FUNCTION "ASW_MAL1S032Ctrl" : VOID
TITLE =MAL1S032 Section control: LINE 1 SEC 32 KILN 1
//COPYRIGHT:    (C) 2009 BY  BUHLER AG
//                           CH-9240 UZWIL  SWITZERLAND
//
//PRODUCT:      WinCoS_BIW01_09
//
//TITLE:        LINE 1 SEC 32 KILN 1
//                 Section control
//
//--------------------------------------------------------------------------------
//
//IDENT:        AUTHOR:             DEPT:                              DATE:
//
//P01_FC832.1.0 K.Renz              CSB41                              09.Okt.2009
//              1st Release
//
//--------------------------------------------------------------------------------
//
//PURPOSE:
//
//REFERENCES : GCSOSMAN
//
//--------------------------------------------------------------------------------
//
//
//0000 to 0999: Main Functions
//              0 =Main Function Cylic
//              1 =Main Function Coldstart/Newstart
//              2 =Main Function Warm Start
AUTHOR : KR
FAMILY : USW
VERSION : 9.9


VAR_INPUT
  InCode : INT ;
END_VAR
VAR_TEMP
  tmpStartNext : BOOL ;	//Condition to Start next element
  tmpFlagFault : BOOL ;	//Flag mechanical fault
  tmpEnableFeed : BOOL ;
  tmpStartScale : BOOL ;
  tmpStartLiqScale : BOOL ;	//Enable to Start Lipquid Scale
  tmpSndBin : INT ;
  tmpRcvBin : INT ;
  tmpBool : BOOL ;
  tmpByte : BYTE ;
  tmpWord : WORD ;
  tmpDWord : DWORD ;
  tmpInt : INT ;
  tmpRET : INT ;
  tmpDInt : DINT ;
  tmpCyclusTime : DINT ;
  tmpWetSteep : BOOL ;
END_VAR
BEGIN
NETWORK
TITLE =
//=================================================
//=================================================
//S T A R T   M A I N   F U N C T I O N
//=================================================
//=================================================
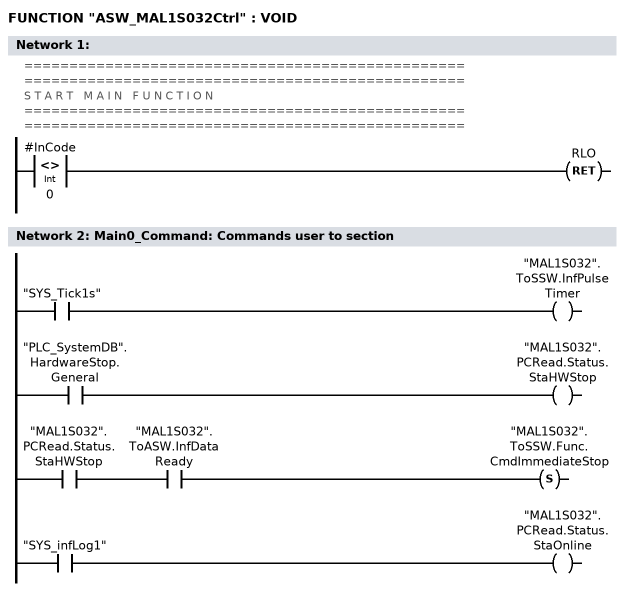
      L     #InCode;
      L     0;
      <>I   ;
      BEB   ;

NETWORK
TITLE =Main0_Command: Commands user to section

      NOP   0;
//-Tick 1 second---
      U     "SYS_Tick1s";
      =     "MAL1S032".ToSSW.InfPulseTimer;
//-Hardware stop---
      U     "PLC_SystemDB".HardwareStop.General;
      =     "MAL1S032".PCRead.Status.StaHWStop;
      U     "MAL1S032".PCRead.Status.StaHWStop;
      U     "MAL1S032".ToASW.InfDataReady;
      S     "MAL1S032".ToSSW.Func.CmdImmediateStop;
//-Online---
      U     "SYS_infLog1";
      =     "MAL1S032".PCRead.Status.StaOnline;
NETWORK
TITLE =ASW_UC: User commands to section

      NOP   0;
//-Additional user commands---
//-GP standard commands---
      AUF   "MAL1S032";
      L     L#0; // Enter the differenz of the target weight and prestop weight
      T     "MAL1S032".VarTemp.InOutValue3; // Prestop weight
      CALL "STD_LineSecStdSub" (
           InCode                   := 2001);// Section function: Standard section commands

//-Condition CmdSequenzStop---
      U     "MAL1S032".ToSSW.Func.CmdSequenzStop;
//      S     "MAL1S032".ToSSW.Func.CmdSequenzStop
      R     "MAL1S032".ToSSW.Func.CmdSequenzStop;
//-Extended section commands---
//      AUF   "MAL1S032"
//      CALL  "STD_LineSecStdSub"
//       InCode:=2002                     // Section function: Extended section commands
//-Status from pulse commands---
      CLR   ;
      =     "MAL1S032".PCRead.ExtFuncOn.Pulse00OverrideLL;
      =     "MAL1S032".PCRead.ExtFuncOn.Pulse01;
      =     "MAL1S032".PCRead.ExtFuncOn.Pulse02;
      =     "MAL1S032".PCRead.ExtFuncOn.Pulse03;
      =     "MAL1S032".PCRead.ExtFuncOn.Pulse04;
      =     "MAL1S032".PCRead.ExtFuncOn.Pulse05;
      =     "MAL1S032".PCRead.ExtFuncOn.Pulse06;
      =     "MAL1S032".PCRead.ExtFuncOn.Pulse07;
//
NETWORK
TITLE =Main0_Dest: Destination
//99 = Undefined Condition
// 0 = Wait to Loading
// 1 = Loading
// 2 = Process Aktive
// 3 = Unloading
// 4 = Cleaning
// 5 = Finish Unloading
// 6 = Process End
// 7 = Cooling Active
// 8 = Wait to Unloading
// 9 =
//10 = Wait for Start Loading
//11 = Start process is not possible! First loading round is not closed!
//12 = Wait for Start Process
//13 = Can not be unloaded! Same batch in previous section!
//14 = Turning is not possible! Srew is not in position!
//15 = Cleaning not finished!
//16 = Process aktive and wait for water! Water not filled!
//17 = Spraying is not possible! Wait for water!
//18 = Cleaning is not possible! Wait for water!
//19 = Automatic function obstructs by active ILO-Mode!
//20 = Automatic startup is breacked! Wait for continue!
//21 = Wait for release unloading!
//22 = Brennerluft zu kalt!   // NEU
      L     99; // Undefined condition

      U     "MAL1S032".PCRead.Step.StPassive;
      UN    "MAL1S032".ToASW.InfDataReady;
      O     ;
      U     "MAL1S032".PCRead.Step.StIdling;
      UN    "MAL1S032".ToASW.InfDataReady;
      SPBN  M300;
      L     0; // Wait for loading
      SPA   M030;
M300: NOP   0;

      U     "MAL1S032".PCRead.Step.StWait;
      U     "MAL1S032".ToASW.InfDataReady;
      SPBN  M310;
      L     10; // Wait for start loading
      SPA   M030;
M310: NOP   0;

      U     "MAL1S032".ToASW.InfDataReady;
      UN    "MAL1S032".PCRead.Step.StWait;
      UN    "MAL1S032".PCRead.Fault.EsMech;
//    UN    "MAL1S006".PCRead.Status.StaAutostart
      U     DB832.DBX  123.0;
      U     DB832.DBX  123.1;
      SPBN  M320;
      L     20; // Automatic startup is breacked! Wait for continue!
      SPA   M030;
M320: NOP   0;

      U     "MAL1S032".PCWrite.ExtFuncOn.StartProcess;
      L     S5T#30S;
      SA    T     86;
      U     T     86;

      U     "MAL1S032".PCRead.Step.StActive;
      U     "MAL1S032Par".Par.FlagFunction_1.StepLoading;
      UN    "MAL1S032Par".Par.FlagProcess.ProcessActive;
      U     "MAL1S032Par".Par.FlagFunction_1.LoadEnd;
      UN    "MAL1S032Par".Par.FlagFunction_1.LoadFirstPartEnd;
// Prozess-Start erst moeglich wenn Darre 2 Schritt 3 beendet hat oder nicht aktiv ist!!
      U(    ;
      U(    ;
      L     "MAL1S033Par".Par.ParIntMachine.ActualStep;
      L     4;
      >=I   ;
      )     ;
      ON    "MAL1S033Par".Par.FlagProcess.ProcessActive;
      )     ;

      SPBN  M311;
      L     11; // Start process is not possible! First loading round is not closed!
      SPA   M030;
M311: NOP   0;

      U     "MAL1S032".ToASW.InfDataReady;
      U(    ;
      O     "MAL1S032".PCRead.Step.StActive;
      O     "MAL1S032".PCRead.Step.StReady;
      )     ;
      U     "MAL1S032Par".Par.FlagFunction_1.FinishLoading;
      U     "G266M".A_3111_MXZ41MA.A_3111_BZS43.StTrue; // sensor zero point
      UN    "MAL1S032Par".Par.FlagProcess.ProcessActive; // Process active
      SPBN  M312;
      L     12; // Wait for start process
      SPA   M030;
M312: NOP   0;

      U     "MAL1S032".ToASW.InfDataReady;
      U     "MAL1S032Par".Par.FlagFunction_1.StepLoading;
      UN    "MAL1S032Par".Par.FlagFunction_1.FinishLoading;
      UN    "MAL1S032Par".Par.FlagProcess.ProcessActive;
      SPBN  M301;
      L     1; // Loading
      SPA   M030;
M301: NOP   0;

      U     "MAL1S032Par".Par.FlagProcess.TurningFloor;
      UN(   ;
      U     "G265M".A_3111_MXZ21_31MA.A_3111_BZS33.InpTrue;
      U     "G265M".A_3111_MXZ21_31MA.A_3111_BZS23.InpTrue;
      )     ;
      SPBN  M314;
      L     14; // Turning is not possible! Srew is not in position!
      SPA   M030;
M314: NOP   0;

      U     "SYS_infLog0";
      SPBN  M317;
      L     17; // Spraying is not possible! Wait for water!
      SPA   M030;
M317: NOP   0;

      U     "G266M".Gr.InManual; // FLOOR DRIVES KILNINGBOX 1
      UN    "G266M".Gr.VarFault; // FLOOR DRIVES KILNINGBOX 1
      U     "G266M".A_3111_MXZ41MA.Ma.StStopped; // FLOOR DRIVES KILNINGBOX 1
      U     "MAL1S032Par".Par.FlagFunction_1.TurningStart;
      U     "MAL1S032Par".Par.FlagProcess.TurningFloor;
      U     "MAL1S032".ToASW.InfDataReady;
      SPBN  M319;
      L     19; // Automatic function obstructs by active ILO-Mode!
      SPA   M030;
M319: NOP   0;

      U     "MAL1S032".Gr.OutSelected[303]; //-->G303M Defroster Flaps Kilningbox
      UN    "MAL1S032Par".Par.FlagProcess2.Schaltp_5;
      U     "MAL1S032Par".Par.FlagProcess.ProcessActive;
      UN    "MAL1S032Par".Par.FlagProcess.Cooling_Activ;
      SPBN  M322;
      L     22; // Brennerluft zu kalt!
      SPA   M030;
M322: NOP   0;

      U     "MAL1S032Par".Par.FlagProcess.ProcessActive;
      UN    "MAL1S032Par".Par.FlagProcess.Cooling_Activ;
      SPBN  M302;
      L     2; // Process aktive
      SPA   M030;
M302: NOP   0;

      U     "MAL1S032".ToASW.InfDataReady;
      UN    "MAL1S034".PCRead.State.StFeeding;
      U     "MAL1S032Par".Par.FlagFunction_1.StepUnloading;
      UN    "MAL1S032Par".Par.FlagFunction_1.FinishUnloading;
      SPBN  M321;
      L     21; // Wait for release unloading!
      SPA   M030;
M321: NOP   0;

      U     "MAL1S032".ToASW.InfDataReady;
      U     "MAL1S032Par".Par.FlagFunction_1.StepUnloading;
      SPBN  M303;
      L     3; // Unloading
      SPA   M030;
M303: NOP   0;

      U     "SYS_infLog0";
      SPBN  M315;
      L     15; // Cleaning not finished!
      SPA   M030;
M315: NOP   0;

      U     "SYS_infLog0";
      SPBN  M318;
      L     18; // Cleaning is not possible! Wait for water!
      SPA   M030;
M318: NOP   0;

      U     "MAL1S032".ToASW.InfDataReady;
      U     "MAL1S032Par".Par.FlagFunction_1.StepCleaning;
      UN    "MAL1S032Par".Par.FlagFunction_1.FinishCleaning;
      SPBN  M304;
      L     4; // Cleaning
      SPA   M030;
M304: NOP   0;

      U     "MAL1S032".ToASW.InfDataReady;
      U     "MAL1S032Par".Par.FlagFunction_1.FinishUnloading;
      UN    "MAL1S032Par".Par.FlagFunction_1.StepCleaning;
      UN    "MAL1S032Par".Par.FlagFunction_1.FinishCleaning;
      SPBN  M305;
      L     5; // Finish unloading
      SPA   M030;
M305: NOP   0;

      U     "SYS_infLog0";
      SPBN  M306;
      L     6; // Process End
      SPA   M030;
M306: NOP   0;

      U     "MAL1S032Par".Par.FlagProcess.ProcessActive; // Process active
      U     "MAL1S032Par".Par.FlagProcess.Cooling_Activ; // Cooling
      SPBN  M307;
      L     7; // Cooling Active
      SPA   M030;
M307: NOP   0;

      U     "MAL1S032".ToASW.InfSameBatchPrevSec;
      U     "MAL1S032".ToASW.InfDataReady;
      U     "MAL1S032Par".Par.FlagProcess.ProcessEnd;
      UN    "MAL1S032Par".Par.FlagProcess.ProcessActive;
      UN    "MAL1S032Par".Par.FlagFunction_1.StepLoading;
      UN    "MAL1S032Par".Par.FlagFunction_1.StepUnloading;
      SPBN  M313;
      L     13; // Can not be unloaded! Same batch in previous section!
      SPA   M030;
M313: NOP   0;

      U     "MAL1S032".ToASW.InfDataReady;
      UN    "MAL1S032".ToASW.InfSameBatchPrevSec;
      U     "MAL1S032Par".Par.FlagProcess.ProcessEnd;
      UN    "MAL1S032Par".Par.FlagProcess.ProcessActive;
      UN    "MAL1S032Par".Par.FlagFunction_1.StepUnloading;
      UN    "MAL1S032Par".Par.FlagFunction_1.FinishUnloading;
      UN    "MAL1S032Par".Par.FlagFunction_1.StepCleaning;
      UN    "MAL1S032Par".Par.FlagFunction_1.FinishCleaning;
      SPBN  M308;
      L     8; // Wait for Unloading
      SPA   M030;
M308: NOP   0;

      U     "SYS_infLog0";
      SPBN  M316;
      L     16; // Process aktive and wait for water! Water not filled!
      SPA   M030;
M316: NOP   0;

M030: T     "MAL1S032Par".SectionStatus;


NETWORK
TITLE =Main0_Next: Ready for next batch

      ON    "MAL1S032".ToASW.InfDataReady;
      =     "MAL1S032".ToSSW.InfReadyForNewBatch;
NETWORK
TITLE =Main0_Control: Control section

      NOP   0;
//-Process commands from PCS---
      AUF   "MAL1S032";
      CALL "GCS7_SecCtrlMain" (// Methode O_Section
           CODE                     := 7);
//-Process commands from user---
      AUF   "MAL1S032";
      CALL "GCS7_SecCtrlMain" (// Methode Control
           CODE                     := 0);
//-Process section step---
      AUF   "MAL1S032";
      CALL "GCS7_SecCtrlMain" (// Methode Step_execute
           CODE                     := 2);
      AUF   "MAL1S032";
      CALL "GCS7_SecCtrlMain" (// Methode Step_transition
           CODE                     := 3);
//-Process section state---
      AUF   "MAL1S032";
      CALL "GCS7_SecCtrlMain" (// Methode State
           CODE                     := 4);

NETWORK
TITLE =Main0_Init: Init

      UN    "MAL1S032".ToASW.Transition.ToWait;
      UN    "MAL1S032".ToASW.CmdNewBatch;
      SPB   in00;
//-User initialization---
      AUF   "MAL1S032";
//
//-Section function: Init ---
      AUF   "MAL1S032";
      CALL "STD_LineSecStdSub" (
           InCode                   := 2003);// Section function: Init
//
//-Group interface---
//
//-Initialise bin objects---
//
//-Emptying job---
      U     "MAL1S032".JobAc.StaBatch.StaEmptyingBatch;
      S     "MAL1S032".PCRead.Status.StaLoaded;
//
//-Error Batch---
//
in00: NOP   0;

NETWORK
TITLE =ASW_VB: Various functions before bin control

      NOP   0;
//
//-Update staSameSndRcv in sender binlist---
NETWORK
TITLE =Main0_GrEMM: Enable manual mode
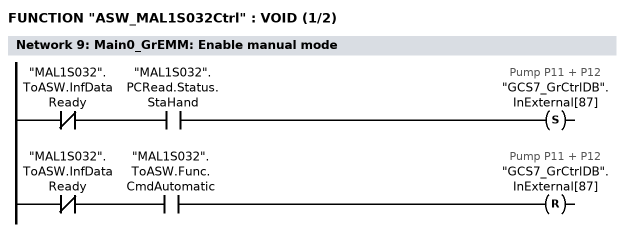

      UN    "MAL1S032".ToASW.InfDataReady;
      U     "MAL1S032".PCRead.Status.StaHand;
      S     "GCS7_GrCtrlDB".InExternal[87]; // Pump P11 + P12

      UN    "MAL1S032".ToASW.InfDataReady;
      U     "MAL1S032".ToASW.Func.CmdAutomatic;
      R     "GCS7_GrCtrlDB".InExternal[87]; // Pump P11 + P12

NETWORK
TITLE =Main0_GrNRS: Not Relevant for started / Fault
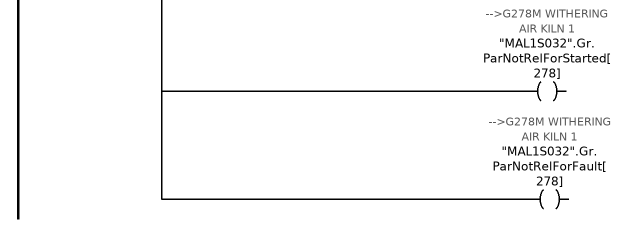

      NOP   0;
      SET   ;
      =     "MAL1S032".Gr.ParNotRelForStarted[1]; //-->G001G Power supply circuit +C11
      =     "MAL1S032".Gr.ParNotRelForFault[1]; //-->G001G Power supply circuit +C11
      =     "MAL1S032".Gr.ParNotRelForStarted[2]; //-->G002G Contactor panel power supply 1
      =     "MAL1S032".Gr.ParNotRelForFault[2]; //-->G002G Contactor panel power supply 1
      =     "MAL1S032".Gr.ParNotRelForStarted[3]; //-->G003G PLC monitoring
      =     "MAL1S032".Gr.ParNotRelForFault[3]; //-->G003G PLC monitoring
      =     "MAL1S032".Gr.ParNotRelForStarted[26]; // -->G026G Alarm horns
      =     "MAL1S032".Gr.ParNotRelForFault[26]; // -->G026G Alarm horns
      =     "MAL1S032".Gr.ParNotRelForStarted[269]; //-->G269M Temperature Mes.  Kilningbox 1
      =     "MAL1S032".Gr.ParNotRelForFault[269]; //-->G269M Temperature Mes.  Kilningbox 1

      U     "MAL1S032Par".Par.FlagFunction_1.StepLoading;
      =     "MAL1S032".Gr.ParNotRelForStarted[271]; //-->G271M FAN KILN 1
      =     "MAL1S032".Gr.ParNotRelForFault[271]; //-->G271M FAN KILN 1
      =     "MAL1S032".Gr.ParNotRelForStarted[272]; //-->G272M FRESH AIR LOUVER KILN 1
      =     "MAL1S032".Gr.ParNotRelForFault[272]; //-->G272M FRESH AIR LOUVER KILN 1
      =     "MAL1S032".Gr.ParNotRelForStarted[273]; //-->G273M RECYCLING AIR LOUVER KILN 1
      =     "MAL1S032".Gr.ParNotRelForFault[273]; //-->G273M RECYCLING AIR LOUVER KILN 1
      =     "MAL1S032".Gr.ParNotRelForStarted[274]; //-->G274M EXHAUST AIR LOUVER KILN 1
      =     "MAL1S032".Gr.ParNotRelForFault[274]; //-->G274M EXHAUST AIR LOUVER KILN 1
      =     "MAL1S032".Gr.ParNotRelForStarted[275]; //-->G275M LOUVER HEATING GLASS TUBE HEAT EXCHANGER
      =     "MAL1S032".Gr.ParNotRelForFault[275]; //-->G275M LOUVER HEATING GLASS TUBE HEAT EXCHANGER
      =     "MAL1S032".Gr.ParNotRelForStarted[276]; //-->G276 MHEATING KILN 1
      =     "MAL1S032".Gr.ParNotRelForFault[276]; //-->G276M HEATING KILN 1
      =     "MAL1S032".Gr.ParNotRelForStarted[277]; //-->G277M LOUVER AIR HEATER 1 FOR KILN 1
      =     "MAL1S032".Gr.ParNotRelForFault[277]; //-->G277M LOUVER AIR HEATER 1 FOR KILN 1
      =     "MAL1S032".Gr.ParNotRelForStarted[278]; //-->G278M WITHERING AIR KILN 1
      =     "MAL1S032".Gr.ParNotRelForFault[278]; //-->G278M WITHERING AIR KILN 1

      NOP   0;

NETWORK
TITLE =Main0_GrSelection: Group selection
// List of the used objects in the section
// ==========================
// G021G       GENERAL ELEMENTS KILN 1
// G284M       BELT CONVEYOR 7100 KILN
// G261M       BELT CONVEYOR 7200 KILN
// G262M       BELT CONVEYOR 7300 KILN
// G263M       BELT CONVEYOR 7301 KILN
// G264M       BELT CONVEYOR 7400 KILN
// G265M       LIFTING DEVICE KILN 1
// G266M       TRAVELLING DRIVE KILN 1
// G267M       UNLOADING / LOADING SCREW KILN 1
// G268M       DISCHARGE DOOR KILN 1
// G269M       TEMPERATURE MES. KILN 1
// G270M       AIR SHUT SLIDE KILN 1
// G271M       FAN KILN 1
// G272M       FRESH AIR LOUVER KILN 1
// G273M       RECYCLING AIR LOUVER KILN 1
// G274M       EXHAUST AIR LOUVER KILN 1
// G275M       LOUVER HEATING GLASS TUBE HEAT EXCHANGER
// G276M       HEATING KILN 1
// G277M       LOUVER AIR HEATER 1 FOR KILN 1
// G278M       WITHERING AIR KILN 1
// G279M       HEATING KILN 1 + 2
// G280M       CHAIN CONVEYOR 9001 KILN 1
// G281M       ELEVATOR 9002 AFTER KILN
// G282M       FLAP BOX 9008
// G283M       CULM BATCH BIN 9005
//
      NOP   0;
//-Condition for preselection---
      U     "MAL1S032".ToASW.InfDataReady;
      SPB   GS01;
//-Deselect groups ---
      CALL "GCS7_GrpCtrlMain" , "GCS7_GrCtrlDBTmp" (// GrCtr.Methode Deselect
           Code                     := 3,
           Sec                      := "MAL1S032".Gr);
      SPA   GS02;
//-Select groups ---
GS01: NOP   0;
//-Prepare for preselection ---
      CALL "GCS7_GrpCtrlMain" , "GCS7_GrCtrlDBTmp" (// GrCtr.Methode Init Preselection
           Code                     := 1,
           Sec                      := "MAL1S032".Gr);
//
//
//-Preselect used groups --
      SET   ;
      S     "MAL1S032".Gr.InPreselect[21]; //-->G021G GENERAL ELEMENTS KILN 1
      S     "MAL1S032".Gr.InPreselect[269]; //-->G269M TEMPERATURE MES. KILN 1

//--- Option
      U     "MAL1S032".PCRead.Step.StActive; // Loading
      O     "MAL1S032".PCRead.Step.StReady; // Process active
      U(    ;
      L     "G269M".A_3191_BTE11.OutValuePc; // AIR TEMPERATURE OUTSIDE
      L     1500; // 15.00°C
      <=I   ;
      )     ;
      UN(   ;
      U     "MAL1S032Par".Par.FlagProcess2.Schaltp_15;
      U     "MAL1S032Par".Par.FlagProcess2.Schaltp_70;
      )     ;
      U     "SYS_infLog0"; // Keine Freigabe!!
      S     "MAL1S032".Gr.InPreselect[276]; //-->G276M HEATING KILN 1
      S     "MAL1S032".Gr.InPreselect[277]; //-->G277M LOUVER AIR HEATER 1 FOR KILN 1
      S     "MAL1S032".Gr.InPreselect[275]; //-->G275M LOUVER HEATING GLASS TUBE HEAT EXCHANGER

// Oeffnen und Schliessen der Defroster-Klappe
      U     "G275M".USW8; // Defrosterklappe AUF
      S     "MAL1S032".Gr.InPreselect[275]; //-->G275M LOUVER HEATING GLASS TUBE HEAT EXCHANGER

//------------------------------Loading kilningbox-----------------------------------
      U     "MAL1S032".PCRead.Step.StActive;
      U     "MAL1S032Par".Par.FlagFunction_1.StepLoading; // Step loading
      S     "MAL1S032".Gr.InPreselect[265]; //-->G265M LIFTING DEVICE KILN 1

      U     "MAL1S032".PCRead.Step.StActive;
      U     "MAL1S032Par".Par.FlagFunction_1.StepLoading; // Step loading
      UN    "MAL1S032Par".Par.FlagFunction_1.FinishLoading; // start process kilning
      S     "MAL1S032".Gr.InPreselect[266]; //-->G266M TRAVELLING DRIVE KILN 1
      S     "MAL1S032".Gr.InPreselect[267]; //-->G267M UNLOADING / LOADING SCREW KILN 1
      S     "MAL1S032".Gr.InPreselect[268]; //-->G268M DISCHARGE DOOR KILN 1
      S     "MAL1S032".Gr.InPreselect[270]; //-->G270M AIR SHUT SLIDE KILN 1
      S     "MAL1S032".Gr.InPreselect[284]; //-->G284M BELT CONVEYOR 7100 KILN
      S     "MAL1S032".Gr.InPreselect[261]; //-->G261M BELT CONVEYOR 7200 KILN
      S     "MAL1S032".Gr.InPreselect[262]; //-->G262M BELT CONVEYOR 7300 KILN
      S     "MAL1S032".Gr.InPreselect[263]; //-->G263M BELT CONVEYOR 7301 KILN
      S     "MAL1S032".Gr.InPreselect[264]; //-->G264M BELT CONVEYOR 7400 KILN

//----------------------------Loading kilningbox finish------------------------------
      U     "MAL1S032".PCRead.Step.StActive;
      O     "MAL1S032".PCRead.Step.StReady;
      U     "MAL1S032Par".Par.FlagProcess.ProcessActive;
      U(    ;
      UN    "G265M".A_3111_MXZ21_31MA.Ma.OutAdjustedLeft;
      ON    "G265M".A_3111_MXZ21_31MA.Ma.OutAdjustedRight;
      )     ;
      S     "MAL1S032".Gr.InPreselect[265]; //-->G265M LIFTING DEVICE KILN 1
//
      U(    ;
      U     "MAL1S032Par".Par.FlagProcess.ProcessActive;
      UN    "MAL1S032Par".Par.FlagFunction_1.StepLoading;
      O     "MAL1S032".PCRead.Step.StReady;
      )     ;
      U     "MAL1S032Par".Par.FlagProcess.ProcessActive;
      U     "MAL1S032Par".Par.FlagProcess.TurningFloor;
      U     "MAL1S032Par".Par.FlagFunction_1.TurningStart;
      S     "MAL1S032".Gr.InPreselect[266]; //-->G266M TRAVELLING DRIVE KILN 1

// Glaettungfahrt zur Parkposition bei Beladen Ende
      U     "MAL1S032Par".Par.FlagProcess.ProcessActive;
      U     "MAL1S032Par".Par.FlagMachine.ImpulsNullstellung;
      S     "MAL1S032".Gr.InPreselect[265]; //-->G265M LIFTING DEVICE KILN 1
      S     "MAL1S032".Gr.InPreselect[266]; //-->G266M TRAVELLING DRIVE KILN 1
      S     "MAL1S032".Gr.InPreselect[267]; //-->G267M UNLOADING / LOADING SCREW KILN 1

//-Cleaning conveyance after loading---
      UN    "MAL1S032Par".Par.FlagFunction_1.StepLoading;
      U     "MAL1S032".PCRead.Step.StReady;
      U     "MAL1S032Par".Par.FlagFunction_0.TimeCleanConvRun;
      S     "MAL1S032".Gr.InPreselect[284]; //-->G284M BELT CONVEYOR 7100 KILN
      S     "MAL1S032".Gr.InPreselect[261]; //-->G261M BELT CONVEYOR 7200 KILN
      S     "MAL1S032".Gr.InPreselect[262]; //-->G262M BELT CONVEYOR 7300 KILN
      S     "MAL1S032".Gr.InPreselect[263]; //-->G263M BELT CONVEYOR 7301 KILN
      S     "MAL1S032".Gr.InPreselect[264]; //-->G264M BELT CONVEYOR 7400 KILN


//-------------------------------Process kilning-------------------------------------
      U     "MAL1S032".PCRead.Step.StActive;
      O     "MAL1S032".PCRead.Step.StReady;
      U     "MAL1S032Par".Par.FlagProcess.ProcessActive; // Process active
      S     "MAL1S032".Gr.InPreselect[268]; //-->G268M DISCHARGE DOOR KILN 1
      S     "MAL1S032".Gr.InPreselect[270]; //-->G270M AIR SHUT SLIDE KILN 1
      S     "MAL1S032".Gr.InPreselect[271]; //-->G271M FAN KILN 1

      U     "MAL1S032".PCRead.Step.StActive;
      O     "MAL1S032".PCRead.Step.StReady;
      U     "MAL1S032Par".Par.FlagProcess.ProcessActive; // Process active
      O     ;
      U     "MAL1S032Par".Par.FlagProcess.ProcessEnd;
      UN    "MAL1S032Par".Par.FlagProcess.ProcessActive;
      UN    "GCS7_GrCtrlDB".InStopped[271]; //-->G271M FAN KILN 1
      S     "MAL1S032".Gr.InPreselect[273]; //-->G273M RECYCLING AIR LOUVER KILN 1
      S     "MAL1S032".Gr.InPreselect[278]; //-->G278M WITHERING AIR KILN 1

      U     "MAL1S032".PCRead.Step.StActive;
      O     "MAL1S032".PCRead.Step.StReady;
      U     "MAL1S032Par".Par.FlagProcess.ProcessActive;
      UN    "MAL1S032Par".Par.FlagProcess.Cooling_Activ;
      S     "MAL1S032".Gr.InPreselect[276]; //-->G276M HEATING KILN 1
      S     "MAL1S032".Gr.InPreselect[277]; //-->G277M LOUVER AIR HEATER 1 FOR KILN 1
      S     "MAL1S032".Gr.InPreselect[279]; //-->G279M HEATING KILN 1 + 2

//--------------------------Kuehlluft-Klappenregelung EIN----------------------------
      U     "MAL1S032".PCRead.Step.StActive;
      O     "MAL1S032".PCRead.Step.StReady;
      U     "MAL1S032Par".Par.FlagProcess.ProcessActive;
      UN    "MAL1S032Par".Par.FlagProcess.Cooling_Activ;
      U     "G272M".USW8; // Klappenregelung Ein
      S     "MAL1S032".Gr.InPreselect[272]; //-->G272M FRESH AIR LOUVER KILN 1

//-------------------------------Process Cooling--------------------------------------
      U     "MAL1S032".PCRead.Step.StActive;
      O     "MAL1S032".PCRead.Step.StReady;
      U     "MAL1S032Par".Par.FlagProcess.ProcessActive;
      U     "MAL1S032Par".Par.FlagProcess.Cooling_Activ;
      O     ;
      U     "MAL1S032Par".Par.FlagProcess.ProcessEnd;
      UN    "MAL1S032Par".Par.FlagProcess.ProcessActive;
      UN    "GCS7_GrCtrlDB".InStopped[271]; //-->G271M FAN KILN 1
      S     "MAL1S032".Gr.InPreselect[272]; //-->G272M FRESH AIR LOUVER KILN 1
      S     "MAL1S032".Gr.InPreselect[277]; //-->G277M LOUVER AIR HEATER 1 FOR KILN 1

//---------------------------Unloading kilning box------------------------------------
      U     "MAL1S032".PCRead.Step.StEmptying;
      U     "MAL1S032Par".Par.FlagFunction_1.StepUnloading; // Step unloading
      U     "MAL1S034".PCRead.State.StFeeding;
      S     "MAL1S032".Gr.InPreselect[268]; //-->G268M DISCHARGE DOOR KILN 1
//
      U     "MAL1S032".PCRead.Step.StEmptying;
      U     "MAL1S032Par".Par.FlagFunction_1.StepUnloading; // Step unloading
      U     "MAL1S034".PCRead.State.StFeeding;
      U     "G268M".Gr.OutEnablePrevGr; //-->G268M DISCHARGE DOOR KILN 1
      S     "MAL1S032".Gr.InPreselect[265]; //-->G265M LIFTING DEVICE KILN 1
//
      U     "MAL1S032".PCRead.Step.StEmptying;
      U     "MAL1S032Par".Par.FlagFunction_1.StepUnloading; // Step unloading
//      UN    "MAL1S032".PCRead.Status.StaTransferOffASW
      U     "G268M".Gr.OutEnablePrevGr; //-->G268M DISCHARGE DOOR KILN 1
      UN    "MAL1S032Par".Par.FlagFunction_1.FinishUnloading;
      U     "MAL1S034".PCRead.State.StFeeding;
      S     "MAL1S032".Gr.InPreselect[267]; //-->G267M UNLOADING / LOADING SCREW KILN 1
//
      U     "MAL1S032".PCRead.Step.StEmptying;
      U     "MAL1S032Par".Par.FlagFunction_1.StepUnloading; // Step unloading
      U     "MAL1S034".PCRead.State.StFeeding;
      UN    "MAL1S032".PCRead.Status.StaTransferOffASW;
      U     "G268M".Gr.OutEnablePrevGr; //-->G268M DISCHARGE DOOR KILN 1
      U     "G267M".Gr.OutEnablePrevGr; //-->G267M UNLOADING / LOADING SCREW KILN 1
      UN    "MAL1S032Par".Par.FlagFunction_0.ScrewAboveProductLayer;
      S     "MAL1S032".Gr.InPreselect[266]; //-->G266M TRAVELLING DRIVE KILN 1
//
// ------------------Parkposition anfahren nach dem Entladen-------------------
//    UN    "MAL1S032Par".Par.FlagFunction_1.StepUnloading
      U     "MAL1S032Par".Par.FlagFunction_1.FinishUnloading;
      U     "MAL1S032Par".Par.FlagMachine.WEGMESSUNG_0;
      S     "MAL1S032".Gr.InPreselect[265]; //-->G265M LIFTING DEVICE KILN 1
      S     "MAL1S032".Gr.InPreselect[266]; //-->G266M TRAVELLING DRIVE KILN 1


//      S     "MAL1S032".Gr.InPreselect[274]    //-->G274M EXHAUST AIR LOUVER KILN 1

//      S     "MAL1S032".Gr.InPreselect[280]    //-->G280M CHAIN CONVEYOR 9001 KILN 1
//      S     "MAL1S032".Gr.InPreselect[281]    //-->G281M ELEVATOR 9002 AFTER KILN
//      S     "MAL1S032".Gr.InPreselect[282]    //-->G282M FLAP BOX 9008
//      S     "MAL1S032".Gr.InPreselect[283]    //-->G283M CULM BATCH BIN 9005
//      L     1
//      L     "MAL1S032Par".StepAct.StepNumber
//      UW
//      ==I                               // step wetsteep
//      =     "MAL1S032Par".Par.FlagGen.WetStep
//
//-Set CmdNewJob ---
      U     "MAL1S032".Gr.InPreselect[284];
      UN    "GCS7_GrCtrlDB".OutOccupied[284];
      S     "G284M".CmdNewJob;
      U     "MAL1S032".Gr.InPreselect[261];
      UN    "GCS7_GrCtrlDB".OutOccupied[261];
      S     "G261M".CmdNewJob;
      U     "MAL1S032".Gr.InPreselect[262];
      UN    "GCS7_GrCtrlDB".OutOccupied[262];
      S     "G262M".CmdNewJob;
      U     "MAL1S032".Gr.InPreselect[263];
      UN    "GCS7_GrCtrlDB".OutOccupied[263];
      S     "G263M".CmdNewJob;
      U     "MAL1S032".Gr.InPreselect[264];
      UN    "GCS7_GrCtrlDB".OutOccupied[264];
      S     "G264M".CmdNewJob;
      U     "MAL1S032".Gr.InPreselect[265];
      UN    "GCS7_GrCtrlDB".OutOccupied[265];
      S     "G265M".CmdNewJob;
      U     "MAL1S032".Gr.InPreselect[266];
      UN    "GCS7_GrCtrlDB".OutOccupied[266];
      S     "G266M".CmdNewJob;
      U     "MAL1S032".Gr.InPreselect[267];
      UN    "GCS7_GrCtrlDB".OutOccupied[267];
      S     "G267M".CmdNewJob;
      U     "MAL1S032".Gr.InPreselect[268];
      UN    "GCS7_GrCtrlDB".OutOccupied[268];
      S     "G268M".CmdNewJob;
      U     "MAL1S032".Gr.InPreselect[269];
      UN    "GCS7_GrCtrlDB".OutOccupied[269];
      S     "G269M".CmdNewJob;
      U     "MAL1S032".Gr.InPreselect[270];
      UN    "GCS7_GrCtrlDB".OutOccupied[270];
      S     "G270M".CmdNewJob;
      U     "MAL1S032".Gr.InPreselect[271];
      UN    "GCS7_GrCtrlDB".OutOccupied[271];
      S     "G271M".CmdNewJob;
      U     "MAL1S032".Gr.InPreselect[272];
      UN    "GCS7_GrCtrlDB".OutOccupied[272];
      S     "G272M".CmdNewJob;
      U     "MAL1S032".Gr.InPreselect[273];
      UN    "GCS7_GrCtrlDB".OutOccupied[273];
      S     "G273M".CmdNewJob;
      U     "MAL1S032".Gr.InPreselect[274];
      UN    "GCS7_GrCtrlDB".OutOccupied[274];
      S     "G274M".CmdNewJob;
      U     "MAL1S032".Gr.InPreselect[275];
      UN    "GCS7_GrCtrlDB".OutOccupied[275];
      S     "G275M".CmdNewJob;
      U     "MAL1S032".Gr.InPreselect[276];
      UN    "GCS7_GrCtrlDB".OutOccupied[276];
      S     "G276M".CmdNewJob;
      U     "MAL1S032".Gr.InPreselect[277];
      UN    "GCS7_GrCtrlDB".OutOccupied[277];
      S     "G277M".CmdNewJob;
      U     "MAL1S032".Gr.InPreselect[278];
      UN    "GCS7_GrCtrlDB".OutOccupied[278];
      S     "G278M".CmdNewJob;
      U     "MAL1S032".Gr.InPreselect[279];
      UN    "GCS7_GrCtrlDB".OutOccupied[279];
      S     "G279M".CmdNewJob;
      U     "MAL1S032".Gr.InPreselect[280];
      UN    "GCS7_GrCtrlDB".OutOccupied[280];
      S     "G280M".CmdNewJob;
      U     "MAL1S032".Gr.InPreselect[281];
      UN    "GCS7_GrCtrlDB".OutOccupied[281];
      S     "G281M".CmdNewJob;
      U     "MAL1S032".Gr.InPreselect[282];
      UN    "GCS7_GrCtrlDB".OutOccupied[282];
      S     "G282M".CmdNewJob;
      U     "MAL1S032".Gr.InPreselect[283];
      UN    "GCS7_GrCtrlDB".OutOccupied[283];
      S     "G283M".CmdNewJob;
//
//
//-Test preselected groups ---
      CALL "GCS7_GrpCtrlMain" , "GCS7_GrCtrlDBTmp" (// GrCtr.Methode Select
           Code                     := 2,
           Sec                      := "MAL1S032".Gr);
//
//-Way conflict if not available---
      CLR   ;
      S     "MAL1S032".Gr.All.OutGrConflict;
//
//-Test occupied real and virtual groups---
GS02: NOP   0;
      U     "MAL1S032".Gr.All.OutSelectionValid;
      UN    "MAL1S032".Gr.All.OutGrIsLocked;
      =     "MAL1S032".Gr.All.InOutASWSelectionOK;
//
//
//----- Send data to selected groups =====
      UN    "MAL1S032".Gr.OutSelected[284]; //G284M
      SPB   GS4;
      L     "MAL1".Para.ParLineNr;
      T     "G284M".Gr.InLine;
GS4:  UN    "MAL1S032".Gr.OutSelected[261]; //G261M
      SPB   GS5;
      L     "MAL1".Para.ParLineNr;
      T     "G261M".Gr.InLine;
GS5:  UN    "MAL1S032".Gr.OutSelected[262]; //G262M
      SPB   GS6;
      L     "MAL1".Para.ParLineNr;
      T     "G262M".Gr.InLine;
GS6:  UN    "MAL1S032".Gr.OutSelected[263]; //G263M
      SPB   GS7;
      L     "MAL1".Para.ParLineNr;
      T     "G263M".Gr.InLine;
GS7:  UN    "MAL1S032".Gr.OutSelected[264]; //G264M
      SPB   GS8;
      L     "MAL1".Para.ParLineNr;
      T     "G264M".Gr.InLine;
GS8:  UN    "MAL1S032".Gr.OutSelected[265]; //G265M
      SPB   GS9;
      L     "MAL1".Para.ParLineNr;
      T     "G265M".Gr.InLine;
GS9:  UN    "MAL1S032".Gr.OutSelected[266]; //G266M
      SPB   GS10;
      L     "MAL1".Para.ParLineNr;
      T     "G266M".Gr.InLine;
GS10: UN    "MAL1S032".Gr.OutSelected[267]; //G267M
      SPB   GS11;
      L     "MAL1".Para.ParLineNr;
      T     "G267M".Gr.InLine;
GS11: UN    "MAL1S032".Gr.OutSelected[268]; //G268M
      SPB   GS12;
      L     "MAL1".Para.ParLineNr;
      T     "G268M".Gr.InLine;
GS12: UN    "MAL1S032".Gr.OutSelected[269]; //G269M
      SPB   GS13;
      L     "MAL1".Para.ParLineNr;
      T     "G269M".Gr.InLine;
GS13: UN    "MAL1S032".Gr.OutSelected[270]; //G270M
      SPB   GS14;
      L     "MAL1".Para.ParLineNr;
      T     "G270M".Gr.InLine;
GS14: UN    "MAL1S032".Gr.OutSelected[271]; //G271M
      SPB   GS15;
      L     "MAL1".Para.ParLineNr;
      T     "G271M".Gr.InLine;
GS15: UN    "MAL1S032".Gr.OutSelected[272]; //G272M
      SPB   GS16;
      L     "MAL1".Para.ParLineNr;
      T     "G272M".Gr.InLine;
GS16: UN    "MAL1S032".Gr.OutSelected[273]; //G273M
      SPB   GS17;
      L     "MAL1".Para.ParLineNr;
      T     "G273M".Gr.InLine;
GS17: UN    "MAL1S032".Gr.OutSelected[274]; //G274M
      SPB   GS18;
      L     "MAL1".Para.ParLineNr;
      T     "G274M".Gr.InLine;
GS18: UN    "MAL1S032".Gr.OutSelected[275]; //G275M
      SPB   GS19;
      L     "MAL1".Para.ParLineNr;
      T     "G275M".Gr.InLine;
GS19: UN    "MAL1S032".Gr.OutSelected[276]; //G276M
      SPB   GS20;
      L     "MAL1".Para.ParLineNr;
      T     "G276M".Gr.InLine;
GS20: UN    "MAL1S032".Gr.OutSelected[277]; //G277M
      SPB   GS21;
      L     "MAL1".Para.ParLineNr;
      T     "G277M".Gr.InLine;
GS21: UN    "MAL1S032".Gr.OutSelected[278]; //G278M
      SPB   GS22;
      L     "MAL1".Para.ParLineNr;
      T     "G278M".Gr.InLine;
GS22: UN    "MAL1S032".Gr.OutSelected[279]; //G279M
      SPB   GS23;
      L     "MAL1".Para.ParLineNr;
      T     "G279M".Gr.InLine;
GS23: UN    "MAL1S032".Gr.OutSelected[280]; //G280M
      SPB   GS24;
      L     "MAL1".Para.ParLineNr;
      T     "G280M".Gr.InLine;
GS24: UN    "MAL1S032".Gr.OutSelected[281]; //G281M
      SPB   GS25;
      L     "MAL1".Para.ParLineNr;
      T     "G281M".Gr.InLine;
GS25: UN    "MAL1S032".Gr.OutSelected[282]; //G282M
      SPB   GS26;
      L     "MAL1".Para.ParLineNr;
      T     "G282M".Gr.InLine;
GS26: UN    "MAL1S032".Gr.OutSelected[283]; //G283M
      SPB   GS27;
      L     "MAL1".Para.ParLineNr;
      T     "G283M".Gr.InLine;
GS27: NOP   0;
NETWORK
TITLE =Main0_GrCmd: CMD section to Groups

      NOP   0;
//-Way Adjust Time---
      O     "MAL1S032".Gr.All.CmdNewSelection;
      O     "MAL1S032".ToASW.CmdModify;
      S     "MAL1S032".ToSSW.CmdNewWay;
      AUF   "MAL1S032";
      CALL "GCS7_SecCtrlMain" (// Methode Adjust Time
           CODE                     := 13);
//-Continue---
      U     "MAL1S032".ToASW.Func.CmdStart;
      O     "MAL1S032".ToASW.Func.CmdNextStep;
      S     "MAL1S032".Gr.All.CmdContinue;
//-Fault reset---
      U     "MAL1S032".ToASW.Func.CmdFaultReset;
      S     "MAL1S032".Gr.All.CmdFaultReset;
//-Manual mode---
      U     "MAL1S032".ToASW.Func.CmdAutomatic;
      S     "MAL1S032".Gr.All.CmdManualOff;
      UN    "MAL1S032".PCRead.Status.StaHand;
      S     "MAL1S032".Gr.All.CmdManualOffRel;
//-Clear idling---
      U     "MAL1S032".PCRead.Status.StaImmediateStopASW;
      S     "MAL1S032".Gr.All.CmdClearIdling;
//-Start next---
      UN    "MAL1S032".PCRead.Status.StaStep;
      O     "MAL1S032".ToASW.Func.CmdNextStep;
      U(    ;
      L     "MAL1S032".PCRead.OutWayAdjustTime;
      L     2;
      >I    ;
      O     "MAL1S032".ToASW.InfWayAdjustTimeEnd;
      )     ;
      UN    "MAL1S032".Gr.All.CmdNewSelection;
      UN    "MAL1S032".PCRead.Step.StWait;
      =     #tmpStartNext; //-->VarStartNext
//-Start next feed---
      U     "MAL1S032".Gr.Wgr.OutStartedRel;
      ON    "MAL1S032".ToASW.InfWayAdjustTimeEnd;
      UN    "MAL1S032".PCRead.Status.StaFeedOffASW;
      UN    "MAL1S032".PCRead.Status.StaImmediateStopASW;
//KR040220100      U     "MAL1S032".Gr.Mgr.OutStartedRel
      U     "MAL1S032".PCRead.Step.StActive;
      =     "MAL1S032".Gr.Feed.InEnable;
      =     #tmpEnableFeed;
      U     #tmpStartNext;
      U     "MAL1S032".Gr.Wgr.OutStartedRel;
      U     "MAL1S032".Gr.All.OutAutoStartOk;
      U     "MAL1S032".PCRead.Status.StaAutostartSec;
      =     "MAL1S032".Gr.Feed.CmdNext;
//-Start next machine group---
      UN    "MAL1S032".PCRead.Status.StaImmediateStopASW;
      =     "MAL1S032".Gr.Mgr.InEnable;
      U     #tmpStartNext;
      =     "MAL1S032".Gr.Mgr.CmdNext;
//-Start next way group---
      UN    "MAL1S032".PCRead.Status.StaImmediateStopASW;
      =     "MAL1S032".Gr.Wgr.InEnable;
      UN    "MAL1S032".PCRead.Status.StaStep;
      O     "MAL1S032".ToASW.Func.CmdNextStep;
      =     "MAL1S032".Gr.Wgr.CmdNext;
//-Start next general group---
      UN    "MAL1S032".PCRead.Status.StaImmediateStopASW;
      =     "MAL1S032".Gr.Ggr.InEnable;
      U     #tmpStartNext;
      =     "MAL1S032".Gr.Ggr.CmdNext;
//-Update command state---
      CALL "GCS7_GrpCtrlMain" , "GCS7_GrCtrlDBTmp" (// GrCtr.Methode UpdateCmdSt
           Code                     := 4,
           Sec                      := "MAL1S032".Gr);

NETWORK
TITLE =Main0_Status: Fault/Status

      NOP   0;
//- Autostart Section---
      UN    "MAL1S032".ToASW.Func.CmdStart;
      O     "MAL1S032".Gr.All.OutAutoStartOk;
      =     "MAL1S032".TimeoutAutostart.EN;
      CALL "GCS7_TON" (
           IN                       := "MAL1S032".TimeoutAutostart.EN,
           PT                       := 10,
           Q                        := "MAL1S032".TimeoutAutostart.Q,
           ET                       := "MAL1S032".TimeoutAutostart.ET);
      U     "MAL1S032".TimeoutAutostart.Q;
      UN    "MAL1S032".Gr.All.OutAutoStartOk;
      R     "MAL1S032".PCRead.Status.StaAutostartSec;
      U     "MAL1S032".ToASW.Func.CmdStart;
      ON    "MAL1S032".ToASW.InfDataReady;
      S     "MAL1S032".PCRead.Status.StaAutostartSec;
//-Stopped---
      UN    "MAL1S032".Gr.Mgr.InEnable;
      U     "MAL1S032".Gr.All.OutStoppedRel;
      O     "MAL1S032".Gr.All.OutStoppedAll;
      UN    "MAL1S032".PCRead.Status.StaStep;
      O     ;
      U     "MAL1S032".Gr.Mgr.OutStoppedRel;
      U     "MAL1S032".PCRead.Status.StaStep;
      =     "MAL1S032".ToSSW.InfStopped;
//-Started---
      U     "MAL1S032".Gr.Mgr.OutStartedRel;
      =     "MAL1S032".ToSSW.InfStarted;
//-Feeding---
      U     "MAL1S032".Gr.Feed.InEnable; //Section without Feed groups
      ON    "MAL1S032".Gr.Feed.OutStoppedAll;
      U     "MAL1S032".Gr.Feed.OutStartedRel;
      =     "MAL1S032".ToSSW.InfFeeding;
//-Autostart---
      U     "MAL1S032".Gr.All.OutAutostartOkAll;
      U     "MAL1S032".PCRead.Status.StaAutostartSec;
      =     "MAL1S032".PCRead.Status.StaAutostart;
//-DPFault---
      U     "MAL1S032".Gr.All.OutDPFault;
      =     "MAL1S032".PCRead.Status.StaDPFault;
      S     "MAL1S032".ToSSW.Func.CmdFeedOff;
//-Startwarning---
      U     "MAL1S032".Gr.All.OutStartwarning;
      =     "MAL1S032".PCRead.Status.StaStartwarning;
//-Way conflict---
      U     "MAL1S032".Gr.All.OutGrConflict;
      =     "MAL1S032".PCRead.Fault.EsWayConflict;
//-Warning---
      U     "MAL1S032".Gr.All.OutWarning;
      =     "MAL1S032".PCRead.Fault.EsWarning;
//-Fault---
      U     "MAL1S032".Gr.All.OutFaultRel;
      FP    "MAL1S032".PCRead.Fault.EsMech;
      S     "MAL1S032".ToSSW.Func.CmdFeedOff;
//-Sender empty---
      CLR   ;
      =     "MAL1S032".PCRead.Fault.EsEmpty; //-->Sec.EsEmpty
//-Receiver full---
      CLR   ;
      =     "MAL1S032".PCRead.Fault.EsFull;

NETWORK
TITLE =Main0_StatusASW: Status from ASW
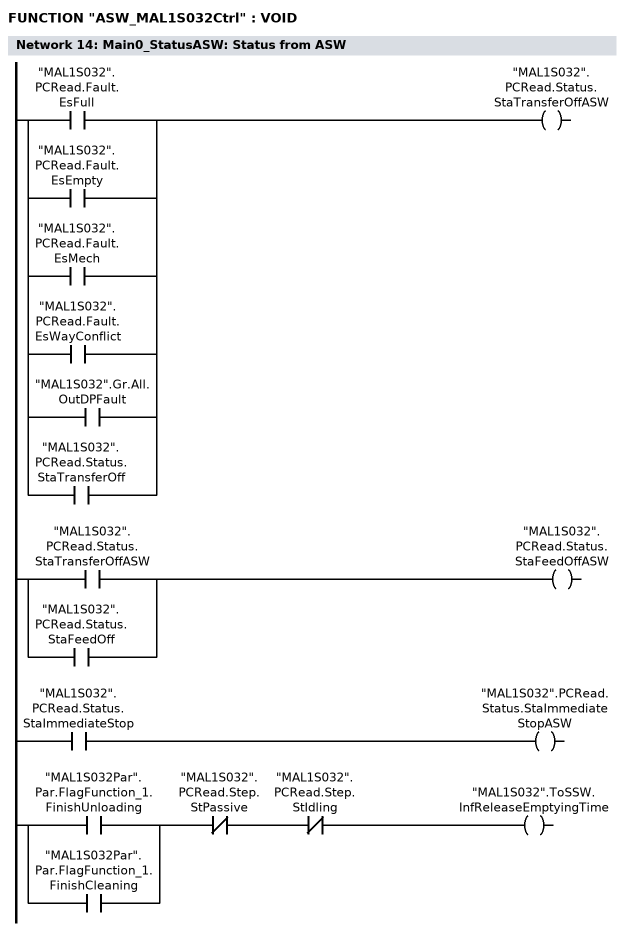

      NOP   0;
//-Transfer off with automatic restart---
      O     "MAL1S032".PCRead.Fault.EsFull;
      O     "MAL1S032".PCRead.Fault.EsEmpty;
      O     "MAL1S032".PCRead.Fault.EsMech;
      O     "MAL1S032".PCRead.Fault.EsWayConflict;
      O     "MAL1S032".Gr.All.OutDPFault;
      O     "MAL1S032".PCRead.Status.StaTransferOff;
      =     "MAL1S032".PCRead.Status.StaTransferOffASW;
//-Feed off with automatic restart---
      U     "MAL1S032".PCRead.Status.StaTransferOffASW;
//      O     "MAL1S032".PCRead.Status.StaEndOfJob
      O     "MAL1S032".PCRead.Status.StaFeedOff;
      =     "MAL1S032".PCRead.Status.StaFeedOffASW;
//-Immediate stop with automatic restart---
      U     "MAL1S032".PCRead.Status.StaImmediateStop;
      =     "MAL1S032".PCRead.Status.StaImmediateStopASW;
//-Emptying time---
      U     "MAL1S032Par".Par.FlagFunction_1.FinishUnloading;
      O     "MAL1S032Par".Par.FlagFunction_1.FinishCleaning;
      UN    "MAL1S032".PCRead.Step.StPassive;
      UN    "MAL1S032".PCRead.Step.StIdling;
      =     "MAL1S032".ToSSW.InfReleaseEmptyingTime;
NETWORK
TITLE =Main0_Transition: Condition for Transition
//      NOP   0
//      NOP   0
////-Active---
//      U     "MAL1S032".Gr.All.InOutASWSelectionOK
//      U     "MAL1S032".PCRead.Step.StWait
//      =     "MAL1S032".ToSSW.CmdGotoActive
////-Ready---
//      U     "MAL1S032".PCRead.Step.StActive
//      UN    "MAL1S032".ToASW.InfSameBatchPrevSec
//      U     "MAL1S032Par".Par.FlagFunction_1.FinishLoading
//      =     "MAL1S032".ToSSW.CmdGotoReady
////-Emptying---
//      U     "MAL1S032".PCRead.Step.StReady
//      UN    "MAL1S032".ToASW.InfSameBatchPrevSec
//      U     "MAL1S032Par".Par.FlagProcess.ProcessEnd
//      UN    "MAL1S032Par".Par.FlagProcess.ProcessActive
//      =     "MAL1S032".ToSSW.CmdGotoEmptying
////-Emptied---
//      U     "MAL1S032".PCRead.Step.StEmptying
//      UN    "MAL1S032".PCRead.Status.StaLoaded
//      U     "MAL1S032Par".Par.FlagFunction_1.FinishCleaning
//      =     "MAL1S032".ToSSW.CmdGotoEmptied
////-Result section---
////-Idling---
//      U     "MAL1S032".PCRead.Step.StEmptied
//      =     "MAL1S032".ToSSW.CmdGotoIdling
////-Passive---
//      U     "MAL1S032".PCRead.Step.StIdling
//      U     "MAL1S032".ToSSW.InfStopped
//      =     "MAL1S032".ToSSW.CmdGotoPassive
//
      NOP   0;
//-Active---
      U     "MAL1S032".Gr.All.InOutASWSelectionOK;
      U     "MAL1S032Par".Par.FlagFunction_1.StepLoading;
      O     ;
      U     "MAL1S032".Gr.All.InOutASWSelectionOK;
      U     "MAL1S032".PCRead.Step.StWait; //KR03022010
      UN    "MAL1S032".SecNom.Par1On.Cmd01; // With Loading
      UN    "MAL1S032".ToASW.InfSameBatchPrevSec;
      =     "MAL1S032".ToSSW.CmdGotoActive;
//-Ready---
      U     "MAL1S032".PCRead.Step.StActive;
//      UN    "MAL1S032".ToASW.InfSameBatchPrevSec
      U     "MAL1S032Par".Par.FlagFunction_1.FinishLoading;
      =     "MAL1S032".ToSSW.CmdGotoReady;
      U     "MAL1S032".ToASW.InfSameBatchPrevSec;
      U     "MAL1S032".PCRead.Step.StActive;
      U     "MAL1S032Par".Par.FlagFunction_1.FinishLoading;
      =     "MAL1S032".SecAc.Sta1On.Inf09; // "SecDB".ToASW.CmdGotoReady
//-Emptying---
      U     "MAL1S032".PCRead.Step.StReady;
//      UN    "MAL1S032".ToASW.InfSameBatchPrevSec
      U     "MAL1S032Par".Par.FlagProcess.ProcessEnd;
      UN    "MAL1S032Par".Par.FlagProcess.ProcessActive;
      =     "MAL1S032".ToSSW.CmdGotoEmptying;

//KR03022010 um in den Status emptying zu gelangen muß 0 als next section für einen
//Zyklus eingetragen werden  --->
      L     834;
      UN    "MAL1S032".ToSSW.CmdGotoEmptying;
      SPB   asse;
      L     0;
asse: T     "MAL1S032".ToSSW.InNextSecDB;
//<---

//KR03022010      U     "MAL1S032".ToASW.InfSameBatchPrevSec
      U     "MAL1S032".PCRead.Step.StReady;
      U     "MAL1S032Par".Par.FlagProcess.ProcessEnd;
      UN    "MAL1S032Par".Par.FlagProcess.ProcessActive;
      =     "MAL1S032".SecAc.Sta1On.Inf10; // "SecDB".ToASW.CmdGotoEmptying
//-Emptied---
      U     "MAL1S032".PCRead.Step.StEmptying;
      UN    "MAL1S032".PCRead.Status.StaLoaded;
      U     "MAL1S032Par".Par.FlagFunction_1.FinishCleaning;
      =     "MAL1S032".ToSSW.CmdGotoEmptied;
//-Result section---
//-Idling---
//KR03022010 damit die Zelle auch später entladen werden kann
      U(    ;
      U     "MAL1S034".PCRead.Step.StActive;
      O     ;
      U     "MAL1S034".ToASW.InfDataReady;
      U     "MAL1S032".PCRead.Step.StWait;
      O(    ; //Sektion hat Jobdaten bekommen
      L     "MAL1S032".JobNom.JobNr;
      L     "MAL1S034".JobNom.JobNr;
      ==D   ;
      )     ;
      )     ;
      U     "MAL1S032".PCRead.Step.StEmptied;
      =     "MAL1S032".ToSSW.CmdGotoIdling;
//-Passive---
      U     "MAL1S032".PCRead.Step.StIdling;
      U     "MAL1S032".ToSSW.InfStopped;
      =     "MAL1S032".ToSSW.CmdGotoPassive;

NETWORK
TITLE =Main0_Move: Move to next section

      NOP   0;
//-------------------------------------------
//-General Condition for move
//-------------------------------------------
//KR03022010      U     "MAL1S032".ToSSW.CmdGotoEmptying
//KR03022010-->
      U(    ;
      U     "MAL1S032".PCRead.Step.StEmptying;
      U     "MAL1S032Par".Par.FlagFunction_1.FinishCleaning;
      )     ;
      O     "MAL1S032".ToSSW.CmdGotoEmptied;
//<---
      O     "MAL1S032".PCRead.Step.StEmptying;
      SPBN  Move;
//->Move batch to section MAL1S034
      AUF   "MAL1S032";
      CALL "GCS7_SecCtrlMain" (// Methode Move Data
           CODE                     := 5);
      UN    "MAL1S032".ToASW.CmdDataMoved;
      SPB   Move;
Move: NOP   0;
NETWORK
TITLE =ASW_AH:Alarm horns

      UN    "MAL1S032".ToASW.Func.CmdHornOn;
      SPB   AHJ1;
      CALL "SYS_Horn_Code" (
           FcCode                   := 1,//Set Alarm
           ParObjectType            := 4000,
           ParObjectNo              := 0,
           ParHornCode              := 98);
AHJ1: UN    "MAL1S032".ToASW.Func.CmdHornOff;
      SPB   AH00;
      CALL "SYS_Horn_Code" (
           FcCode                   := 2,//Reset Alarm
           ParObjectType            := 4000,
           ParObjectNo              := 0,
           ParHornCode              := 1);
      CALL "SYS_Horn_Code" (
           FcCode                   := 2,//Reset Alarm
           ParObjectType            := 4000,
           ParObjectNo              := 0,
           ParHornCode              := 10);
      CALL "SYS_Horn_Code" (
           FcCode                   := 2,//Reset Alarm
           ParObjectType            := 4000,
           ParObjectNo              := 0,
           ParHornCode              := 11);
      CALL "SYS_Horn_Code" (
           FcCode                   := 2,//Reset Alarm
           ParObjectType            := 4000,
           ParObjectNo              := 0,
           ParHornCode              := 12);
AH00: NOP   0;
NETWORK
TITLE =ASW_FT: Feeding Time

      AUF   "MAL1S032";
      CALL "STD_LineSecStdSub" (
           InCode                   := 2004);// Section function: Feeding time

NETWORK
TITLE =ASW_OL: Override low level
//
      AUF   "MAL1S032";
//
      NOP   0;
NETWORK
TITLE =ASW_VA: VA Various functions after section control
//       AUF   "MAL1S032"
//// Copy bin number to section DB
//      L     "MAL1S032".JobAc.BatchSndBin
//      L     "MAL1S032".MAL1S001SND33.Ingr[1].Bin
//      T     "MAL1S032".JobAc.BatchSndBin
//      <>I
//      S     "MAL1S032".ChangeBit.CBit1
////
//      L     "MAL1S032".JobAc.BatchRcvBin
//      L     "MAL1S032".MAL1S001RCV34.Ingr[1].Bin
//      T     "MAL1S032".JobAc.BatchRcvBin
//      <>I
//      S     "MAL1S032".ChangeBit.CBit1
////
//      L     "MAL1S032".JobAc.BatchRcvBin
//      L     "MAL1S032".MAl1S034RCV36.Ingr[1].Bin
//      T     "MAL1S032".JobAc.BatchRcvBin
//      <>I
//      S     "MAL1S032".ChangeBit.CBit1
////
//      L     "MAL1S032".JobAc.BatchSndBin
//      L     "MAL1S032".MAl1S034SND35.Ingr[1].Bin
//      T     "MAL1S032".JobAc.BatchSndBin
//      <>I
//      S     "MAL1S032".ChangeBit.CBit1
////
//


NETWORK
TITLE =ASW_EJ End of job

      NOP   0;
//
//-Fluidlift monitoring---
NETWORK
TITLE =ASW_VE: VE New value event
//
//-Group interface---
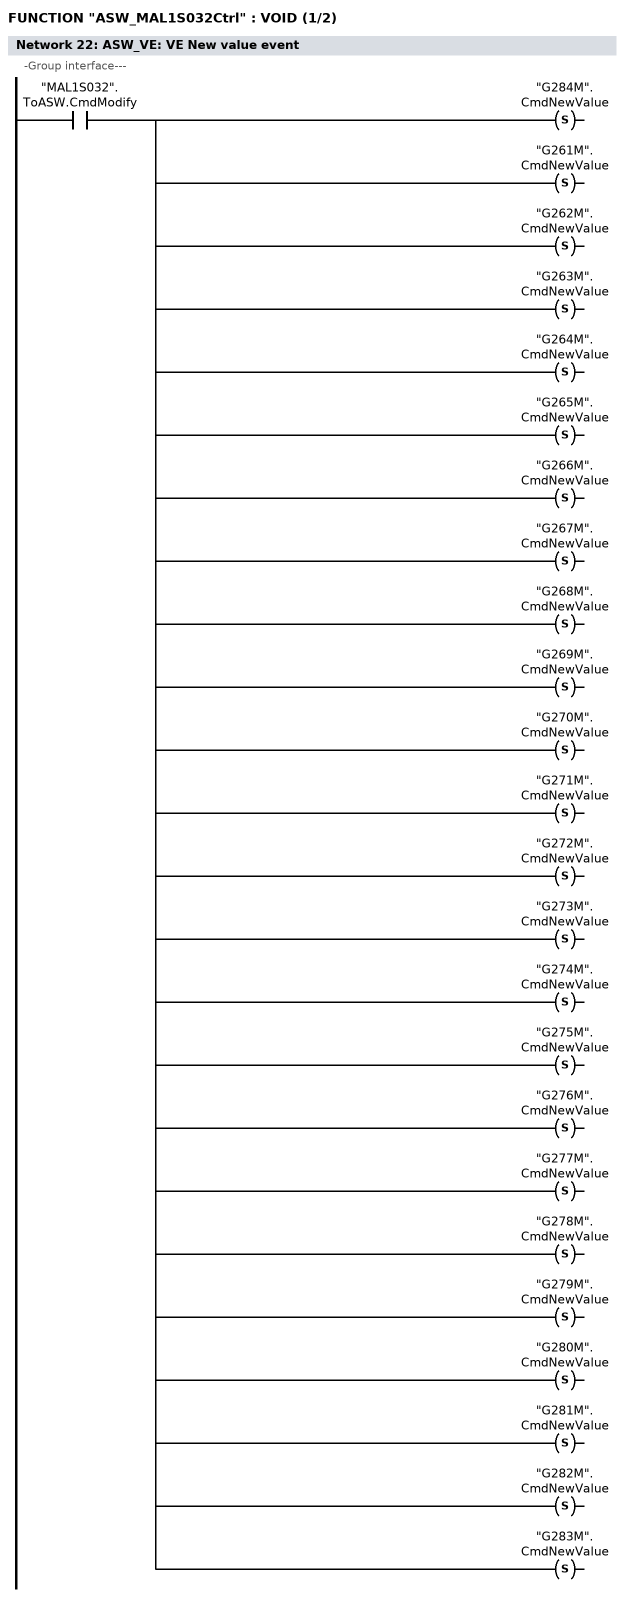
      U     "MAL1S032".ToASW.CmdModify;
      S     "G284M".CmdNewValue;
      S     "G261M".CmdNewValue;
      S     "G262M".CmdNewValue;
      S     "G263M".CmdNewValue;
      S     "G264M".CmdNewValue;
      S     "G265M".CmdNewValue;
      S     "G266M".CmdNewValue;
      S     "G267M".CmdNewValue;
      S     "G268M".CmdNewValue;
      S     "G269M".CmdNewValue;
      S     "G270M".CmdNewValue;
      S     "G271M".CmdNewValue;
      S     "G272M".CmdNewValue;
      S     "G273M".CmdNewValue;
      S     "G274M".CmdNewValue;
      S     "G275M".CmdNewValue;
      S     "G276M".CmdNewValue;
      S     "G277M".CmdNewValue;
      S     "G278M".CmdNewValue;
      S     "G279M".CmdNewValue;
      S     "G280M".CmdNewValue;
      S     "G281M".CmdNewValue;
      S     "G282M".CmdNewValue;
      S     "G283M".CmdNewValue;


NETWORK
TITLE =ASW_NV: New value data



NETWORK
TITLE =ASW_WJ: Weight job
//
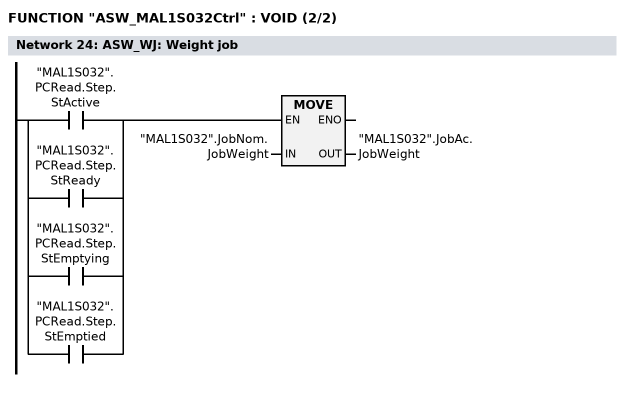
      U     "MAL1S032".PCRead.Step.StActive;
      O     "MAL1S032".PCRead.Step.StReady;
      O     "MAL1S032".PCRead.Step.StEmptying;
      O     "MAL1S032".PCRead.Step.StEmptied;
      SPBN  WJ08;
//
      L     "MAL1S032".JobNom.JobWeight; //Target/Actual registration if no scale
      T     "MAL1S032".JobAc.JobWeight;
//
WJ08: NOP   0;
//--------------------------------------------
//PW Prestop weight
//--------------------------------------------
      NOP   0;
NETWORK
TITLE =ASW_SC: Section status text and colour
//
      AUF   "MAL1S032";
      CALL "STD_LineSecStdSub" (
           InCode                   := 2055);// Section function: WinCoS.SectionInfoCode
//
NETWORK
TITLE =ASW_5010: Prepare Log-Data cyclic
// Prepare Log-Data cyclic
      U     "MAL1S032".ToASW.InfDataReady; // job in section
      U     M      4.7; // scan 30sec
      SPBN  N501;
      AUF   "MAL1S032";
      L     0;
      T     #tmpInt;
      CALL "SIEMENS_FILL" (
           BVAL                     := #tmpInt,
           RET_VAL                  := #tmpRET,
           BLK                      := "SSA_LOG_Value_Queue".Input);
// header
//
      L     B#16#1E; // type 30 = kilning
      T     "SSA_LOG_Value_Queue".Input.Header.SecType; // type
      L     B#16#1; // format 1 = cyclic
      T     "SSA_LOG_Value_Queue".Input.Header.Format; // format
      L     "MAL1S032".JobNom.JobNr;
      T     "SSA_LOG_Value_Queue".Input.Para_0005;
      L     "MAL1ProcessTime".Sektion_32.Gesamtzeit_in_Minuten;
      T     "SSA_LOG_Value_Queue".Input.Para_0007;
      L     "MAL1S032Par".Par.ParIntMachine.ActualStep;
      T     "SSA_LOG_Value_Queue".Input.Para_0008;
      L     "MAL1S032Par".ActTimeStepProcess.SteptimeActMinOverall;
      T     "SSA_LOG_Value_Queue".Input.Para_0009;
//
// values doubleword
//=================================
      L     "G269M".A_3191_BTE07.OutValueUnits; // AIR TEMPERATURE ABOVE FLOOR
      T     "SSA_LOG_Value_Queue".Input.Para_0015;
//=================================
      L     "G269M".A_3191_BTE10.OutValueUnits; // act value before heater
      T     "SSA_LOG_Value_Queue".Input.Para_0017;
//=================================
      L     "G269M".A_3191_BTE01.OutValueUnits; // AIR TEMPERATURE BELOW FLOOR
      T     "SSA_LOG_Value_Queue".Input.Para_0019;
//=================================
//P4 setpoint from SCAD
      L     "MAL1S032Par".StepAct.TemperaturBelowFloor; // setpoint from SCADA
      T     "SSA_LOG_Value_Queue".Input.Para_0021;
//=================================
      L     "G269M".A_3191_BTE11.OutValueUnits; // AIR TEMPERATURE AMBIENT AIR
      T     "SSA_LOG_Value_Queue".Input.Para_0023;
//=================================
      L     "G269M".A_3191_BTE05.OutValueUnits; // act value temperature in diffusor fan 1
      T     "SSA_LOG_Value_Queue".Input.Para_0025;
//=================================
      L     "G269M".A_3191_BTE08.OutValueUnits; // act value temperature after burner 1
      T     "SSA_LOG_Value_Queue".Input.Para_0027;
//=================================
      L     "G269M".A_3191_BTE12.OutValueUnits; // act value temperature after heat exchanger flap
      T     "SSA_LOG_Value_Queue".Input.Para_0029;
//=================================
      L     0; // act value airpressure after heatexchanger
      T     "SSA_LOG_Value_Queue".Input.Para_0031;
//=================================
      L     0; // act value product temperature lowpoint
      T     "SSA_LOG_Value_Queue".Input.Para_0033;
//=================================
      L     0; // act value product temperature middlepoint
      T     "SSA_LOG_Value_Queue".Input.Para_0035;
//=================================
      L     0; // act value product temperature highpoint
      T     "SSA_LOG_Value_Queue".Input.Para_0037;
//=================================
      L     0; // act value steam flowrate
      T     "SSA_LOG_Value_Queue".Input.Para_0039;
//=================================
      L     "G273M".A_3135_MXZ11.OutPosition; // LOUVER RECYCLE AIR 1
      ITD   ;
      T     "SSA_LOG_Value_Queue".Input.Para_0041;
//=================================
      L     "G273M".A_3136_MXZ11.OutPosition; // LOUVER RECYCLE AIR 2
      ITD   ;
      T     "SSA_LOG_Value_Queue".Input.Para_0043;
//=================================
      L     "G272M".A_3150_MXZ11.OutPosition; // LOUVER FRESH AIR 1
      ITD   ;
      T     "SSA_LOG_Value_Queue".Input.Para_0045;
//=================================
      L     0; // act value temperature steam inlet heatexchanger 2
      T     "SSA_LOG_Value_Queue".Input.Para_0047;
//=================================
      L     0; // act position valve1 steam inlet heatexchanger 1
      T     "SSA_LOG_Value_Queue".Input.Para_0049;
//=================================
      L     "G278M".A_3145_MXZ11.OutPosition; // LOUVER WITHERING AIR 1
      ITD   ;
      T     "SSA_LOG_Value_Queue".Input.Para_0051;
//=================================
      L     0;
      T     "SSA_LOG_Value_Queue".Input.Para_0053;
//=================================
      L     0;
      T     "SSA_LOG_Value_Queue".Input.Para_0055;
//=================================
      L     0; // act value position exhaust air flap
      T     "SSA_LOG_Value_Queue".Input.Para_0057;
//=================================
      L     "G277M".A_3140_MXZ11.OutPosition; // LOUVER AIR 1 HEATER
      ITD   ;
      T     "SSA_LOG_Value_Queue".Input.Para_0059;
//=================================
      L     "G277M".A_3141_MXZ11.OutPosition; // LOUVER AIR 2 HEATER
      ITD   ;
      T     "SSA_LOG_Value_Queue".Input.Para_0061;
//=================================
      L     0; // act value position exhaust air flap
      T     "SSA_LOG_Value_Queue".Input.Para_0063;
//=================================
      L     0; // act value position fresh air flap
      T     "SSA_LOG_Value_Queue".Input.Para_0065;
//=================================
      L     "G271M".A_3125_TSC01_AF.OutValueUnits; // ACT. FREQUENCY FAN 1 FU
      T     "SSA_LOG_Value_Queue".Input.Para_0067;
//=================================
      L     "G271M".A_3126_TSC01_AF.OutValueUnits; // ACT. FREQUENCY FAN 2 FU
      T     "SSA_LOG_Value_Queue".Input.Para_0069;
//=================================
      L     "G271M".A_3125_BTE05.OutValueUnits; // TEMPERATURE BEARING TEMPERATUR SENSOR
      L     L#10;
      /D    ;
      T     "SSA_LOG_Value_Queue".Input.Para_0071;
//=================================
      L     "G271M".A_3125_BTE06.OutValueUnits; // TEMPERATURE BEARING TEMPERATUR SENSOR
      L     L#10;
      /D    ;
      T     "SSA_LOG_Value_Queue".Input.Para_0073;
//=================================
      L     "G271M".A_3125_KCU04AI1.OutValueUnits; // VIBRATION MONITOR FAN 1 CHANNEL 1
      L     L#10;
      /D    ;
      T     "SSA_LOG_Value_Queue".Input.Para_0075;
//=================================
      L     "G271M".A_3125_KCU04AI2.OutValueUnits; // VIBRATION MONITOR FAN 1 CHANNEL 2
      L     L#10;
      /D    ;
      T     "SSA_LOG_Value_Queue".Input.Para_0077;
//=================================
      L     "G271M".A_3126_BTE05.OutValueUnits; // TEMPERATURE BEARING TEMPERATUR SENSOR
      L     L#10;
      /D    ;
      T     "SSA_LOG_Value_Queue".Input.Para_0079;
//=================================
      L     "G271M".A_3126_BTE06.OutValueUnits; // TEMPERATURE BEARING TEMPERATUR SENSOR
      L     L#10;
      /D    ;
      T     "SSA_LOG_Value_Queue".Input.Para_0081;
//=================================
      L     "G271M".A_3126_KCU04AI1.OutValueUnits; // VIBRATION MONITOR FAN 2 CHANNEL 1
      L     L#10;
      /D    ;
      T     "SSA_LOG_Value_Queue".Input.Para_0083;
//=================================
      L     "G271M".A_3126_KCU04AI2.OutValueUnits; // VIBRATION MONITOR FAN 2 CHANNEL 2
      L     L#10;
      /D    ;
      T     "SSA_LOG_Value_Queue".Input.Para_0085;
//=================================
      L     0; // spare
      T     "SSA_LOG_Value_Queue".Input.Para_0087;
// values integer
//
      L     L#0; // spare
      T     "SSA_LOG_Value_Queue".Input.Para_0089;
      U     "SYS_infLog0"; // spare
      L     1;
      SPB   MP90;
      L     0;
MP90: T     "SSA_LOG_Value_Queue".Input.Para_0090;
      U     "SYS_infLog0"; // spare
      L     1;
      SPB   MP91;
      L     0;
MP91: T     "SSA_LOG_Value_Queue".Input.Para_0091;
      U     "SYS_infLog0"; // spare
      L     1;
      SPB   MP92;
      L     0;
MP92: T     "SSA_LOG_Value_Queue".Input.Para_0092; // spare
      U     "SYS_infLog0"; // spare
      L     1;
      SPB   MP93;
      L     0;
MP93: T     "SSA_LOG_Value_Queue".Input.Para_0093; // spare
      U     "SYS_infLog0"; // cleaning on/off
      L     1;
      SPB   MP94;
      L     0;
MP94: T     "SSA_LOG_Value_Queue".Input.Para_0094; // spare
      U     "SYS_infLog0"; // spare
      L     1;
      SPB   MP95;
      L     0;
MP95: T     "SSA_LOG_Value_Queue".Input.Para_0095; // spare
      U     "SYS_infLog0"; // spare
      L     1;
      SPB   MP96;
      L     0;
MP96: T     "SSA_LOG_Value_Queue".Input.Para_0096; // spare
      U     "MAL1S032Par".Par.FlagProcess.TurningFloor; // turning floor 0/1
      L     1;
      SPB   MP97;
      L     0;
MP97: T     "SSA_LOG_Value_Queue".Input.Para_0097; //  turning floor 0/1
      U     "MAL1S032Par".Par.FlagProcess.Cooling_Activ; // cooling down 0/1
      L     1;
      SPB   MP98;
      L     0;
MP98: T     "SSA_LOG_Value_Queue".Input.Para_0098; // cooling down 0/1
      NOP   0;
      NOP   0;
// cont log-messages
      L     "SSA_LOG_Value_Queue".Input.Para_0099; // message counter
      L     1;
      +I    ;
      T     "SSA_LOG_Value_Queue".Input.Para_0099; // message counter

// put timestamp into message
      CALL "SIEMENS_BLKMOV" (
           SRCBLK                   := "MAL1ProcessTime".Arbeitsbereich.dt2,
           RET_VAL                  := #tmpInt,
           DSTBLK                   := "SSA_LOG_Value_Queue".Input.TimeStamp);
//
      CALL "SSA_MH_LogEntry_ActValue" (
           DBNumber                 := 1005);
N501: NOP   0;
NETWORK
TITLE =ASW_5030: Prepare Log-Data step values

      NOP   0;
      NOP   0;
//
// load actual values into average input
// 1. Value
      L     "G269M".A_3191_BTE07.OutValuePc; // AIR TEMPERATURE ABOVE FLOOR
      T     "MAL1S032StepValues".LogValues[1].Wert;
// 2. Value
      L     "G269M".A_3191_BTE01.OutValuePc; // AIR TEMPERATURE BELOW FLOOR
      T     "MAL1S032StepValues".LogValues[2].Wert;
// 3. Value
      L     "G272M".A_3150_MXZ11.OutPosition; // ACT. FRESH AIR
      T     "MAL1S032StepValues".LogValues[3].Wert;
// 4. Value
      L     "G273M".A_3135_MXZ11.OutPosition; // ACT. RECYCLE AIR
      T     "MAL1S032StepValues".LogValues[4].Wert;
// 5. Value
      L     "G271M".A_3125_TSC01_AF.OutValuePc; // ACT. FREQUENCY FAN 1 FU
      T     "MAL1S032StepValues".LogValues[5].Wert;
// 6. Value
      L     "G271M".A_3126_TSC01_AC.Par.OutMonTimeH; // ACT. FREQUENCY FAN 2 FU
      T     "MAL1S032StepValues".LogValues[6].Wert;
// 7. Value
      L     0;
      T     "MAL1S032StepValues".LogValues[7].Wert;
// 8. Value
      L     0;
      T     "MAL1S032StepValues".LogValues[8].Wert;
// 9. Value
      L     0;
      T     "MAL1S032StepValues".LogValues[9].Wert;
// 10. Value
      L     0;
      T     "MAL1S032StepValues".LogValues[10].Wert;
// 11. Value
      L     0;
      T     "MAL1S032StepValues".LogValues[11].Wert;
// 12. Value
      L     0;
      T     "MAL1S032StepValues".LogValues[12].Wert;
      NOP   0;
// Entry Values
      CALL "SSA_MH_Step_Values" , "MAL1S032StepValues" (
           Class                    := B#16#1E,
           InJobNo                  := "MAL1S032".JobNom.JobNr,
           InSectionNumber          := "MAL1S032".Para.ParSecNr,
           InTimeAct                := "MAL1S032Par".ActTimeStepProcess.SteptimeActMinOverall,
           InStepNr                 := "MAL1S032Par".StepAct.StepNumber,
           InProcessMinutes         := "MAL1S032Par".Processtime.Min);

NETWORK
TITLE =ASW_5060: Prepare Log-Data events

      NOP   0;
// load events into event input

// 1. event Process active
      U     "MAL1S032Par".Par.FlagProcess.ProcessActive;
      =     DB2062.DBX  142.1;
      L     1;
      T     DB2062.DBW  274;
// 2. event InfDataReady
      U     "MAL1S032".ToASW.InfDataReady;
      =     DB2062.DBX  142.2;
      L     2;
      T     DB2062.DBW  272;
// 3. event old/new step stopped/started
      L     "MAL1S032Par".Par.ParIntMachine.ActualStep;
      L     1;
      ==I   ;
      U     "MAL1S032Par".Par.FlagProcess.ProcessActive;
      O(    ;
      L     "MAL1S032Par".Par.ParIntMachine.ActualStep;
      L     "MAL1S032Par".Par.ProcessValue.StepNrActCopy;
      ==I   ;
      U(    ;
      L     "MAL1S032Par".Par.ParIntMachine.ActualStep;
      L     1;
      >I    ;
      )     ;
      )     ;
      =     DB2062.DBX  142.3;
      L     3;
      T     DB2062.DBW  270;
// 11. event
      U     "MAL1S032Par".Par.FlagFunction_1.StepLoading; // Step loading
      =     DB2062.DBX  143.3;
      L     1001;
      T     DB2062.DBW  254;
// 12. event Loading Round 1
      U     "MAL1S032Par".Par.FlagFunction_1.StepLoading;
      U(    ;
      L     "G266M".A_3111_MXZ41MA.Ma.OutCntRound;
      L     L#0;
      ==D   ;
      )     ;
      =     DB2062.DBX  143.4;
      L     1003;
      T     DB2062.DBW  252;
// 13. event Loading Round 2
      U     "MAL1S032Par".Par.FlagFunction_1.StepLoading;
      U(    ;
      L     "G266M".A_3111_MXZ41MA.Ma.OutCntRound;
      L     L#1;
      ==D   ;
      )     ;
      =     DB2062.DBX  143.5;
      L     1004;
      T     DB2062.DBW  250;
// 14. event Loading Round 3
      U     "MAL1S032Par".Par.FlagFunction_1.StepLoading;
      U(    ;
      L     "G266M".A_3111_MXZ41MA.Ma.OutCntRound;
      L     L#2;
      ==D   ;
      )     ;
      =     DB2062.DBX  143.6;
      L     1005;
      T     DB2062.DBW  248;
// 15. event Loading Round 4
      U     "MAL1S032Par".Par.FlagFunction_1.StepLoading;
      U(    ;
      L     "G266M".A_3111_MXZ41MA.Ma.OutCntRound;
      L     L#3;
      ==D   ;
      )     ;
      =     DB2062.DBX  143.7;
      L     1006;
      T     DB2062.DBW  246;
// 16. event Loading Round 5
      U     "MAL1S032Par".Par.FlagFunction_1.StepLoading;
      U(    ;
      L     "G266M".A_3111_MXZ41MA.Ma.OutCntRound;
      L     L#4;
      ==D   ;
      )     ;
      =     DB2062.DBX  144.0;
      L     1007;
      T     DB2062.DBW  244;
// 17. event Loading Round 6
      U     "MAL1S032Par".Par.FlagFunction_1.StepLoading;
      U(    ;
      L     "G266M".A_3111_MXZ41MA.Ma.OutCntRound;
      L     L#5;
      ==D   ;
      )     ;
      =     DB2062.DBX  144.1;
      L     1008;
      T     DB2062.DBW  242;
// 18. event  Program withering/kilning
      U     "MAL1S032Par".Par.FlagProcess.ProcessActive;
      =     DB2062.DBX  144.2;
      L     1043;
      T     DB2062.DBW  240;
// 19. event ILO-Mode
      U     "MAL1S032".SecAc.Sta1On.Inf08; // ILO-Mode Section
      =     DB2062.DBX  144.3;
      L     1026;
      T     DB2062.DBW  238;
// 20. event Unloading
      U     "MAL1S032Par".Par.FlagFunction_1.StepUnloading;
      =     DB2062.DBX  144.4;
      L     1020;
      T     DB2062.DBW  236;
// 21. event Unloading Round 1
      U     "MAL1S032Par".Par.FlagFunction_1.StepUnloading;
      U(    ;
      L     "G266M".A_3111_MXZ41MA.Ma.OutCntRound;
      L     L#0;
      ==D   ;
      )     ;
      =     DB2062.DBX  144.5;
      L     1053;
      T     DB2062.DBW  234;
// 22. event Unloading Round 2
      U     "MAL1S032Par".Par.FlagFunction_1.StepUnloading;
      U(    ;
      L     "G266M".A_3111_MXZ41MA.Ma.OutCntRound;
      L     L#1;
      ==D   ;
      )     ;
      =     DB2062.DBX  144.6;
      L     1054;
      T     DB2062.DBW  232;
// 23. event Unloading Round 3
      U     "MAL1S032Par".Par.FlagFunction_1.StepUnloading;
      U(    ;
      L     "G266M".A_3111_MXZ41MA.Ma.OutCntRound;
      L     L#2;
      ==D   ;
      )     ;
      =     DB2062.DBX  144.7;
      L     1055;
      T     DB2062.DBW  230;
// 24. event
      U     "SYS_infLog0";
      =     DB2062.DBX  145.0;
      L     114;
      T     DB2062.DBW  228;
// 25. event Cleaning finished
      U     "MAL1S032Par".Par.FlagFunction_1.FinishCleaning;
      =     DB2062.DBX  145.1;
      L     1032;
      T     DB2062.DBW  226;
// 26. event  Cooling active
      U     "MAL1S032Par".Par.FlagProcess.Cooling_Activ;
      =     DB2062.DBX  145.2;
      L     1037;
      T     DB2062.DBW  224;
// 27. event  Process end
      U     "MAL1S032Par".Par.FlagProcess.ProcessEnd;
      =     DB2062.DBX  145.3;
      L     1038;
      T     DB2062.DBW  222;
// 28. event
      U     "SYS_infLog0";
      =     DB2062.DBX  145.4;
      L     118;
      T     DB2062.DBW  220;
// 29. event
      U     "SYS_infLog0";
      =     DB2062.DBX  145.5;
      L     119;
      T     DB2062.DBW  218;
// 30. event  steam regulator 1 on
      U     "SYS_infLog0";
      =     DB2062.DBX  145.6;
      L     1067;
      T     DB2062.DBW  216;
// 31. event  steam regulator 2 on
      U     "SYS_infLog0";
      =     DB2062.DBX  145.7;
      L     1068;
      T     DB2062.DBW  214;
// 32. event  steam regulator 3 on
      U     "SYS_infLog0";
      =     DB2062.DBX  146.0;
      L     1069;
      T     DB2062.DBW  212;
// 33. event  steam regulator 4 on
      U     "SYS_infLog0";
      =     DB2062.DBX  146.1;
      L     1070;
      T     DB2062.DBW  210;
// 34. event
      U     "SYS_infLog0";
      =     DB2062.DBX  146.2;
      L     124;
      T     DB2062.DBW  208;
// 35. event
      U     "SYS_infLog0";
      =     DB2062.DBX  146.3;
      L     125;
      T     DB2062.DBW  206;
// 36. event
      U     "SYS_infLog0";
      =     DB2062.DBX  146.4;
      L     126;
      T     DB2062.DBW  204;
// 37. event
      U     "SYS_infLog0";
      =     DB2062.DBX  146.5;
      L     127;
      T     DB2062.DBW  202;
// 38. event
      U     "SYS_infLog0";
      =     DB2062.DBX  146.6;
      L     128;
      T     DB2062.DBW  200;
// 39. event
      U     "SYS_infLog0";
      =     DB2062.DBX  146.7;
      L     129;
      T     DB2062.DBW  198;
// 40. event
      U     "SYS_infLog0";
      =     DB2062.DBX  147.0;
      L     130;
      T     DB2062.DBW  196;
//
// 41. event
      U     "SYS_infLog0";
      =     DB2062.DBX  147.1;
      L     131;
      T     DB2062.DBW  194;
// 42. event
      U     "SYS_infLog0";
      =     DB2062.DBX  147.2;
      L     132;
      T     DB2062.DBW  192;
// 43. event
      U     "SYS_infLog0";
      =     DB2062.DBX  147.3;
      L     133;
      T     DB2062.DBW  190;
// 44. event
      U     "SYS_infLog0";
      =     DB2062.DBX  147.4;
      L     134;
      T     DB2062.DBW  188;
// only for test
// 47. event
      U     "SYS_infLog0";
      =     DB2062.DBX  147.7;
      L     47;
      T     DB2062.DBW  182;

// copy data for event-logging
      L     "MAL1ProcessTime".Sektion_32.Gesamtzeit_in_Minuten;
      T     "MAL1S032Par".Processtime.Spare_93;
      L     "MAL1S032Par".Par.ParIntMachine.ActualStep;
      T     "MAL1S032Par".ActTimeStepProcess.Spare_85;

//
      CALL "SSA_MH_EventsToPIC" , DB  2062 (
           CallingSection           := 832,
           ParameterDB_in           := 922,
           MessageTyp               := 30,
           ActTimeStepProcess       := "MAL1S032Par".ActTimeStepProcess,
           Processtime              := "MAL1S032Par".Processtime);
NETWORK
TITLE =ASW_6000: Start process kilning

      U     "MAL1S032".ToASW.InfDataReady;
      U(    ;
      O     "MAL1S032".PCRead.Step.StActive;
      O     "MAL1S032".PCRead.Step.StReady;
      )     ;
      UN    "MAL1S032Par".Par.FlagProcess.ProcessActive;
      U     "MAL1S032Par".Par.FlagFunction_1.FinishLoading;
      U     "MAL1S032".PCWrite.ExtFuncOn.StartProcess; // PIC command "start process kilning"
// Prozess-Start erst moeglich wenn Darre 2 Schritt 3 beendet hat oder nicht aktiv ist!!
      U(    ;
      U(    ;
      L     "MAL1S033Par".Par.ParIntMachine.ActualStep;
      L     4;
      >=I   ;
      )     ;
      ON    "MAL1S033Par".Par.FlagProcess.ProcessActive;
      )     ;

      SPBN  e605;
      SET   ;
      S     "MAL1S032Par".Par.FlagProcess.ProcessActive;
      R     "MAL1S032Par".Par.FlagFunction_1.StepLoading;
      S     "MAL1S032Par".Par.FlagMachine.ImpulsNullstellung;
e605: NOP   0;
//
      U     "MAL1S032Par".Par.FlagProcess.ProcessActive;
      U     "MAL1S032Par".Par.FlagFunction_1.FinishLoading;
      U     "MAL1S032".PCRead.Step.StReady;
      R     "MAL1S032Par".Par.FlagFunction_1.FinishLoading;
//
      U     "MAL1S032Par".Par.FlagProcess.ProcessActive;
      FP    "MAL1S032Par".Par.FlagProcess.StartProzess_FP;
      =     "MAL1S032Par".Par.FlagProcess.StartProzess_SCAN;

// Planieren bis zur Parkposition (0°-Sensor)
      U     "MAL1S032Par".Par.FlagProcess.StartProzess_SCAN;
      SPBN  TAL;
      SET   ;
      S     "MAL1S032Par".Par.FlagMachine.CmdTurnFwdAfterLoading;
TAL:  NOP   0;

//-Cleaning conveyance after loading---
      U     "MAL1S032Par".Par.FlagProcess.StartProzess_SCAN;
      SPBN  CCAL;
      L     "MAL1S032Par".Par.ParIntProcess.TargetTimeCleaning;
      T     "MAL1S032Par".Par.ParIntProcess.ActualTimeCleaning;
CCAL: NOP   0;
      L     "MAL1S032Par".Par.ParIntProcess.ActualTimeCleaning;
      L     0;
      >I    ;
      U(    ; // Nicht vor oder beim Beladen
      U     "MAL1S032".PCRead.Step.StReady;
      UN    "MAL1S032Par".Par.FlagFunction_1.StepLoading;
      )     ;
      UN(   ;
      U     "MAL1S032".PCRead.Step.StReady;
      UN    "MAL1S032".SecNom.Par1On.Cmd01; // With Loading
      UN    "MAL1S032".ToASW.InfSameBatchPrevSec;
      )     ;
      =     "MAL1S032Par".Par.FlagFunction_0.TimeCleanConvRun;


      U     "GCS7_GrCtrlDB".InStarted[270]; //-->G270M AIR SHUT SLIDE KILN 1
      U     "GCS7_GrCtrlDB".InStarted[284]; //-->G284M BELT CONVEYOR 7100 KILN
      U     "GCS7_GrCtrlDB".InStarted[261]; //-->G261M BELT CONVEYOR 7200 KILN
      U     "GCS7_GrCtrlDB".InStarted[262]; //-->G262M BELT CONVEYOR 7300 KILN
      U     "GCS7_GrCtrlDB".InStarted[263]; //-->G263M BELT CONVEYOR 7301 KILN
      U     "GCS7_GrCtrlDB".InStarted[264]; //-->G264M BELT CONVEYOR 7400 KILN
      U     "MAL1S032Par".Par.FlagFunction_0.TimeCleanConvRun;
      U     "SYS_Scan0_Tick1min";
      SPBN  tcc;
      L     "MAL1S032Par".Par.ParIntProcess.ActualTimeCleaning;
      L     -1;
      +I    ;
      T     "MAL1S032Par".Par.ParIntProcess.ActualTimeCleaning;
tcc:  NOP   0;
      U     "MAL1S032Par".Par.FlagFunction_1.StepLoading;
      SPBN  tcc0;
      L     0;
      T     "MAL1S032Par".Par.ParIntProcess.ActualTimeCleaning;
tcc0: NOP   0;

NETWORK
TITLE =ASW_6020: Copy recipe-data in Parameter DB
//
// Clear content recipe in buffer
      L     0;
      T     #tmpInt;
      CALL "SIEMENS_FILL" (
           BVAL                     := #tmpInt,
           RET_VAL                  := #tmpRET,
           BLK                      := "MAL1S032Par".RecipeHeader);
//
      U     "MAL1S032".ToASW.InfDataReady;
      SPBN  No10;
// Copy step loading,unloading,cleaning to parameterDB
      CALL "SIEMENS_BLKMOV" (
           SRCBLK                   := "MAL1S032".SecNom.KILN1.RecipeHeader.Loading,
           RET_VAL                  := "MAL1S032Par".Par.Error.Value,
           DSTBLK                   := "MAL1S032Par".RecipeHeader.Loading);
      CALL "SIEMENS_BLKMOV" (
           SRCBLK                   := "MAL1S032".SecNom.KILN1.RecipeHeader.Unloading,
           RET_VAL                  := "MAL1S032Par".Par.Error.Value,
           DSTBLK                   := "MAL1S032Par".RecipeHeader.Unloading);
      CALL "SIEMENS_BLKMOV" (
           SRCBLK                   := "MAL1S032".SecNom.KILN1.RecipeHeader.Cleaning,
           RET_VAL                  := "MAL1S032Par".Par.Error.Value,
           DSTBLK                   := "MAL1S032Par".RecipeHeader.Cleaning);
//      SPA   E607
No10: NOP   0;
      U     "MAL1S032Par".Par.FlagProcess.ProcessActive;
      SPBN  E607;
// Copy common parameter
      CALL "SIEMENS_BLKMOV" (
           SRCBLK                   := "MAL1S032".SecNom.KILN1.RecipeHeader,
           RET_VAL                  := "MAL1S032Par".Par.Error.Value,
           DSTBLK                   := "MAL1S032Par".RecipeHeader);
//
// Copy step parameter
      U(    ;
      L     "MAL1S032Par".Par.ParIntMachine.ActualStep;
      L     1;
      <I    ;
      )     ;
      O(    ;
      L     "MAL1S032Par".Par.ParIntMachine.ActualStep;
      L     "MAL1S032Par".RecipeHeader.NumberOfSteps;
      >I    ;
      )     ;
      SPB   E607; // error wrong step number
      CALL "SYS_Copy_Array_Element" (
           Source                   := "MAL1S032".SecNom.KILN1.Step,
           Destination              := "MAL1S032Par".StepAct,
           Index                    := "MAL1S032Par".Par.ParIntMachine.ActualStep,
           Fault                    := "MAL1S032Par".Par.Error.Bit);
E607: NOP   0;
NETWORK
TITLE =ASW_6010: Process Kilning Active
//      U     "MAL1S032".ToASW.InfDataReady
//      SPB   NoCl
//// Clear process time in buffer
//      L     0
//      T     "MAL1S032Par".ActTimeStepProcess.SteptimeActHour
//      T     "MAL1S032Par".ActTimeStepProcess.SteptimeActMin
//      T     "MAL1S032Par".ActTimeStepProcess.SteptimeActMinOverall
//      T     "MAL1S032Par".Processtime.Day
//      T     "MAL1S032Par".Processtime.Hour
//      T     "MAL1S032Par".Processtime.Min
//      T     "MAL1S032Par".Processtime.ProcessTimeActive
//      L     L#0                         // clear actual step time
//      T     "MAL1S032Par".Par.ProcessValue.StepTimeAct    // in ms
//NoCl: NOP   0
//// Clear process time in buffer end
//      U     "MAL1S032Par".Par.FlagProcess.ProcessActive
//      SPBN  E606
////-Actual process time---
//      U     "MAL1S032Par".Par.FlagProcess.StartProzess_SCAN
//      SPBN  actk
//      L     1                           // Start process first step
//      T     "MAL1S032Par".Par.ParIntMachine.ActualStep
//      T     "MAL1S032Par".Par.ProcessValue.StepNrActCopy
//      SPA   neSk
//actk: NOP   0
//// Prozesszeit
//      L     "MAL1ProcessTime".Sektion_32.Tage
//      INC   1                           // malters do not accept day 0!!
//      T     "MAL1S032Par".Processtime.Day
//      L     "MAL1ProcessTime".Sektion_32.Stunden
//      T     "MAL1S032Par".Processtime.Hour    // Processtime in h
//      L     "MAL1ProcessTime".Sektion_32.Minuten
//      T     "MAL1S032Par".Processtime.Min    // Processtime in min
//      U     "MAL1ProcessTime".Sektion_32.Prozess_aktiv    // active bit section
//2
//      L     1
//      SPB   nTa
//      L     0
//nTa:  T     "MAL1S032Par".Processtime.ProcessTimeActive
//// Test new step
//      L     "MAL1S032Par".Par.ParIntMachine.ActualStep
//      L     "MAL1S032Par".Par.ProcessValue.StepNrActCopy
//      ==I
//      SPB   olSk
//neSk: NOP   0
//      L     "MAL1S032Par".Par.ParIntMachine.ActualStep
//      T     "MAL1S032Par".Par.ProcessValue.StepNrActCopy
////
//      L     L#0                         // clear actual step time
//      T     "MAL1S032Par".Par.ProcessValue.StepTimeAct    // in ms
//      L     0
//      T     "MAL1S032Par".ActTimeStepProcess.SteptimeActMinOverall    //
//Steptime in min overall
////
//      U(
//      L     "MAL1S032Par".Par.ParIntMachine.ActualStep
//      L     DB922.DBW 1500
//      >I
//      )
//      SPB   Pedk                        // last step is finished
//      SET
//      S     "MAL1S032StepValues".StartStep    // start step for average
//calculating
//      SPA   E606                        // to secure, that new step-data are
//copied
//olSk: NOP   0
//      L     "ASW_GraphicData".General.CycleTime[1].Actual
//      T     #tmpCyclusTime
//
//      U     "G271M".A_3125_MXZ01MA.Ma.StStartedFwd    // min one fan must run
//      O     DB371.DBX 1411.2            // min one fan must run
//      UN    "G269M".A_3191_BTE07.OutOverflow    //AIR TEMPERATURE ABOVE FLOOR
//      UN    "G269M".A_3191_BTE07.OutFaultAI    //AIR TEMPERATURE ABOVE FLOOR
//      UN    "G269M".A_3191_BTE01.OutOverflow    //AIR TEMPERATURE BELOW FLOOR
//      UN    "G269M".A_3191_BTE01.OutFaultAI    //AIR TEMPERATURE BELOW FLOOR
//      SPBN  NoTi                        // count steptime only when fan running
//and sensor alive
//      L     "MAL1S032Par".Par.ProcessValue.StepTimeAct    // in ms
//      L     #tmpCyclusTime
//      +D
//      T     "MAL1S032Par".Par.ProcessValue.StepTimeAct    // in ms
//NoTi: NOP   0
//      L     "MAL1S032Par".Par.ProcessValue.StepTimeAct    // in ms
//      L     L#86400000                  // ms/d
//      MOD
//      L     L#3600000                   // ms/h
//      /D
//      T     "MAL1S032Par".ActTimeStepProcess.SteptimeActHour    // Steptime in h
//
//      L     "MAL1S032Par".Par.ProcessValue.StepTimeAct
//      L     L#3600000                   // ms/h
//      MOD
//      L     L#60000                     // ms/min
//      /D
//      T     "MAL1S032Par".ActTimeStepProcess.SteptimeActMin    // Steptime in
//min
//
//      L     "MAL1S032Par".Par.ProcessValue.StepTimeAct
//      L     L#60000                     // ms/min
//      /D
//      T     "MAL1S032Par".ActTimeStepProcess.SteptimeActMinOverall    //
//Steptime in min overall
//
      U     "MAL1S032".ToASW.InfDataReady;
      SPB   NoCl;
// Clear process time in buffer
      L     0;
      T     "MAL1S032Par".ActTimeStepProcess.SteptimeActHour;
      T     "MAL1S032Par".ActTimeStepProcess.SteptimeActMin;
      T     "MAL1S032Par".ActTimeStepProcess.SteptimeActMinOverall;
      T     "MAL1S032Par".Processtime.Day;
      T     "MAL1S032Par".Processtime.Hour;
      T     "MAL1S032Par".Processtime.Min;
      T     "MAL1S032Par".Processtime.ProcessTimeActive;
      L     L#0; // clear actual step time
      T     "MAL1S032Par".Par.ProcessValue.StepTimeAct; // in ms
NoCl: NOP   0;
// Clear process time in buffer end
      U     "MAL1S032Par".Par.FlagProcess.ProcessActive;
      SPBN  E606;
//-Actual process time---
      U     "MAL1S032Par".Par.FlagProcess.StartProzess_SCAN;
      SPBN  actk;
      L     1; // Start process first step
      T     "MAL1S032Par".Par.ParIntMachine.ActualStep;
      T     "MAL1S032Par".Par.ProcessValue.StepNrActCopy;
      SPA   neSk;
actk: NOP   0;
// Prozesszeit
      L     "MAL1ProcessTime".Sektion_32.Tage;
      INC   1; // malters do not accept day 0!!
      T     "MAL1S032Par".Processtime.Day;
      L     "MAL1ProcessTime".Sektion_32.Stunden;
      T     "MAL1S032Par".Processtime.Hour; // Processtime in h
      L     "MAL1ProcessTime".Sektion_32.Minuten;
      T     "MAL1S032Par".Processtime.Min; // Processtime in min
      U     "MAL1ProcessTime".Sektion_32.Prozess_aktiv; // active bit section 24
      L     1;
      SPB   nTa;
      L     0;
nTa:  T     "MAL1S032Par".Processtime.ProcessTimeActive;
// Test new step
      L     "MAL1S032Par".Par.ParIntMachine.ActualStep;
      L     "MAL1S032Par".Par.ProcessValue.StepNrActCopy;
      ==I   ;
      SPB   olSk;
neSk: NOP   0;
      L     "MAL1S032Par".Par.ParIntMachine.ActualStep;
      T     "MAL1S032Par".Par.ProcessValue.StepNrActCopy;
//
      L     L#0; // clear actual step time
      T     "MAL1S032Par".Par.ProcessValue.StepTimeAct; // in ms
      L     0;
      T     "MAL1S032Par".ActTimeStepProcess.SteptimeActMinOverall; // Steptime in min overall
      SET   ; //JV161209 ===>
      R     "MAL1S032Par".Par.FlagProcess.Inf04; // Zeitauswertung aktiv
//JV161209 <===
//
      U(    ;
      L     "MAL1S032Par".Par.ParIntMachine.ActualStep;
      L     "MAL1S032Par".RecipeHeader.NumberOfSteps;
      >I    ;
      )     ;
      U(    ;
      L     "MAL1S032Par".Par.ParIntMachine.ActualStep;
      L     0;
      <>I   ;
      )     ;
      U(    ;
      L     "MAL1S032Par".RecipeHeader.NumberOfSteps;
      L     0;
      >I    ;
      )     ;
      SPB   Pedk; // last step is finished
//      SET   ;
//      S     "MAL1S032StepValues".StartStep; // start step for average calculating
      SPA   E606; // to secure, that new step-data are copied
olSk: NOP   0;
//JV161209      L     "ASW_GraphicData".General.CycleTime[1].Actual
//JV161209      T     #tmpCyclusTime

      U     "G271M".A_3125_MXZ01MA.Ma.StStartedFwd; // min one fan must run
      O     DB371.DBX 1445.2; // min one fan must run
      UN    "G269M".A_3191_BTE07.OutOverflow; //LUFTTEMPERATUR ÜBER DER HORDE
      UN    "G269M".A_3191_BTE07.OutFaultAI; //LUFTTEMPERATUR ÜBER DER HORDE
      UN    "G269M".A_3191_BTE01.OutOverflow; //LUFTTEMPERATUR UNTER DER HORDE
      UN    "G269M".A_3191_BTE01.OutFaultAI; //LUFTTEMPERATUR UNTER DER HORDE
      SPBN  NoTi; // count steptime only when fan running and sensor alive
//JV161209      L     "MAL1S032Par".Par.ProcessValue.StepTimeAct    // in ms
//JV161209      L     #tmpCyclusTime
//JV161209      +D
//JV161209      T     "MAL1S032Par".Par.ProcessValue.StepTimeAct    // in ms
//--Create actual Timeinterval for counting steptime new JV151209 ===>

      CALL "SIEMENS_READ_CLK" (
           RET_VAL                  := MW   200,
           CDT                      := "MAL1S032Par".Par.ProcessValue.ActualTime);

      U     "MAL1S032Par".Par.FlagProcess.Inf04; // Zeitauswertung aktiv
      SPB   diff;
      CALL "SIEMENS_READ_CLK" (
           RET_VAL                  := MW   200,
           CDT                      := "MAL1S032Par".Par.ProcessValue.ActualTimePreviousScan);// Start-Zeit CPU-Clock aktuelle Auswertung
      SET   ;
      S     "MAL1S032Par".Par.FlagProcess.Inf04; // Zeitauswertung aktiv

diff: NOP   0;

      CALL "SB_DT_DT" (
           DT1                      := "MAL1S032Par".Par.ProcessValue.ActualTime,// momentane Zeit CPU-Clock
           DT2                      := "MAL1S032Par".Par.ProcessValue.ActualTimePreviousScan,// Start-Zeit CPU-Clock aktuelle Auswertung
           RET_VAL                  := "MAL1S032Par".Par.ProcessValue.Afeesttijd);// Zeitdifferenz in ms


      L     "MAL1S032Par".Par.ProcessValue.Afeesttijd; // Zeitdifferenz in ms
      L     L#10000; // 10sec
      >=D   ;
      R     "MAL1S032Par".Par.FlagProcess.Inf04; // Zeitauswertung aktiv
      FP    "MAL1S032Par".Par.FlagProcess.Inf05;
      SPBN  NoST;
      L     "MAL1S032Par".Par.ProcessValue.Afeesttijd; // Zeitdifferenz in ms
      SPM   Korr; //JV161209 Da hat wer an der Uhr gedreht.....
      L     L#10150; // 10sec + 150ms  als Maximalüberwachung
      >D    ; //JV161209 Da hat wer an der Uhr gedreht.....
      SPBN  AlOK;
Korr: NOP   0;
      L     L#10000; // 10sec als Grundwert, wenn die Zeit verstellt wurde
      T     "MAL1S032Par".Par.ProcessValue.Afeesttijd; // Zeitdifferenz in ms
AlOK: NOP   0;
      L     "MAL1S032Par".Par.ProcessValue.Afeesttijd; // Zeitdifferenz in ms
      L     "ASW_GraphicData".General.CycleTime[1].Actual; // aktuelle Zykluszeit als Korrektur
      +D    ;
      L     "MAL1S032Par".Par.ProcessValue.StepTimeAct; // in ms
      +D    ;
      T     "MAL1S032Par".Par.ProcessValue.StepTimeAct; // in ms
NoST: NOP   0;
//--Create actual Timeinterval for counting steptime new JV151209 <===

      SPA   OKTi; //JV161209
NoTi: NOP   0;
      SET   ; //JV161209 ===>
      R     "MAL1S032Par".Par.FlagProcess.Inf04; // Zeitauswertung aktiv
//JV161209 <===
OKTi: NOP   0; //JV161209
      L     "MAL1S032Par".Par.ProcessValue.StepTimeAct; // in ms
      L     L#86400000; // ms/d
      MOD   ;
      L     L#3600000; // ms/h
      /D    ;
      T     "MAL1S032Par".ActTimeStepProcess.SteptimeActHour; // Steptime in h

      L     "MAL1S032Par".Par.ProcessValue.StepTimeAct;
      L     L#3600000; // ms/h
      MOD   ;
      L     L#60000; // ms/min
      /D    ;
      T     "MAL1S032Par".ActTimeStepProcess.SteptimeActMin; // Steptime in min

      L     "MAL1S032Par".Par.ProcessValue.StepTimeAct;
      L     L#60000; // ms/min
      /D    ;
      T     "MAL1S032Par".ActTimeStepProcess.SteptimeActMinOverall; // Steptime in min overall

//
// Next Step
//
//   Switch over to next step under conditions:
//   or Maximal steptime
//   or Minimal steptime
//           and
//               or no setpoint delta temp
//               or atual value delta temp is ge setpoint deltatemp
//                   and sensor is ok
//           and
// /              or no setpoint max temp above floor
//              or atual value max temp above floor is ge setpoint max temp above floor
//                  and sensor is ok
// 1 Kriterium
      U(    ;
      L     "MAL1S032Par".ActTimeStepProcess.SteptimeActMinOverall; // Steptime in min overall
      L     "MAL1S032Par".StepAct.StepTime_Max; // Target steptime actual step
      >=I   ;
      )     ;
      O(    ;
// 2 Kriterium
      O(    ;
      U(    ;
      L     "MAL1S032Par".StepAct.DeltaTempSwitchpointStep;
      L     0;
      >=D   ;
      )     ;
// condition, if analogue input is not damaaged   //
      UN    "G269M".A_3191_BTE07.OutOverflow; //AIR TEMPERATURE ABOVE FLOOR
      UN    "G269M".A_3191_BTE07.OutFaultAI; //AIR TEMPERATURE ABOVE FLOOR
      UN    "G269M".A_3191_BTE01.OutOverflow; //AIR TEMPERATURE BELOW FLOOR
      UN    "G269M".A_3191_BTE01.OutFaultAI; //AIR TEMPERATURE BELOW FLOOR
      U(    ;
      L     "G269M".A_3191_BTE01.OutValueUnits; // act value temperature below floor
      L     "G269M".A_3191_BTE07.OutValueUnits; // act value temperature above floor
      -D    ; // delta temp actual
      L     L#10;
      /D    ;
      L     "MAL1S032Par".StepAct.DeltaTempSwitchpointStep;
      <D    ;
      )     ;
      )     ;
// 3 Kriterium
      O(    ;
      U(    ;
      L     "MAL1S032Par".StepAct.MaxTempAboveFloorStep;
      L     L#0; // 0,0°C is illegally switchpoint for max. temperature
      >D    ;
      )     ;
// condition, if analogue input is not damaaged   // MW R2.1
      UN    "G269M".A_3191_BTE01.OutOverflow; //AIR TEMPERATURE BELOW FLOOR
      UN    "G269M".A_3191_BTE01.OutFaultAI; //AIR TEMPERATURE BELOW FLOOR
      U(    ;
      L     "G269M".A_3191_BTE07.OutValueUnits; // act value temperature above floor
      L     L#10;
      /D    ;
      L     "MAL1S032Par".StepAct.MaxTempAboveFloorStep;
      >=D   ;
      )     ;
      )     ;
// 4 Kriterium
// and min. time
      U(    ;
      L     "MAL1S032Par".ActTimeStepProcess.SteptimeActMinOverall; // Steptime in min overall
      L     "MAL1S032Par".StepAct.StepTime_Min; // Target steptime actual step
      >=I   ;
      )     ;
      )     ;
// and not cooling                                // UK 22.01.07
      UN    "MAL1S032Par".Par.FlagProcess.Cooling_Activ;
// 5 Kriterium
      O(    ;
      U     "MAL1S032Par".Par.FlagProcess.Cooling_Activ;
      U(    ;
      L     "G269M".A_3191_BTE07.OutValueUnits; // act value temperature above floor
      L     L#10;
      /D    ;
      L     "MAL1S032Par".StepAct.TemperaturAboveFloor;
      <=D   ;
      )     ;
      O(    ;
      L     "MAL1S032Par".Par.ParIntMachine.ActualStep;
      L     25; // max. 24 Schritte
      >=I   ;
      )     ;
      )     ;
// and min. time
      U(    ;
      L     "MAL1S032Par".ActTimeStepProcess.SteptimeActMinOverall; // Steptime in min overall
      L     "MAL1S032Par".StepAct.StepTime_Min; // Target steptime actual step
      >=I   ;
      )     ;
      SPBN  E606;
// send average step data to PIC
      SET   ;
      S     "MAL1S032StepValues".SendData; // send average step data to PIC
// Next step
      L     "MAL1S032Par".Par.ParIntMachine.ActualStep;
      L     "MAL1S032Par".RecipeHeader.NumberOfSteps;
      >I    ;
      SPB   Pedk; // Last step is finished
//
      L     "MAL1S032Par".Par.ParIntMachine.ActualStep;
      L     1;
      +I    ;
      T     "MAL1S032Par".Par.ParIntMachine.ActualStep;
      L     0;
      T     "MAL1S032Par".ActTimeStepProcess.SteptimeActMinOverall; // Steptime in min Overall
      SPA   E606;
Pedk: NOP   0; // Process has finished
      SET   ;
      R     "MAL1S032Par".Par.FlagProcess.ProcessActive;
      R     "MAL1S032Par".Par.FlagProcess.Cooling_Activ;
      S     "MAL1S032Par".Par.FlagProcess.ProcessEnd;
//
      L     0; // clear step number
      T     "MAL1S032Par".Par.ParIntMachine.ActualStep;
      T     "MAL1S032Par".StepAct.StepNumber;
E606: NOP   0;
NETWORK
TITLE =ASW_6080: Active step kilning
//
      U     "MAL1S032Par".Par.FlagProcess.ProcessActive;
      SPBN  E608;
// copy stepnr for visu
      L     "MAL1S032Par".Par.ParIntMachine.ActualStep;
      T     "MAL1S032Par".Par.ParIntProcess.ActualStep;
// basic speed  fans
      L     "MAL1S032Par".StepAct.SpeedVentilatorBasic;
      T     "MAL1S032Par".Par.ParIntProcess.SpeedVentilatorBasic;
// basic position waste air flaps
      L     "MAL1S032Par".StepAct.PosExhaustAirFlapBasic; // setpoint from recipe
      L     10; // convert to 0.1%
      *I    ;
      T     "MAL1S032Par".Par.ParIntProcess.PosExhaustAirFlapBasic;
// basic position withering air channel flaps
      L     "MAL1S032Par".StepAct.PosWitheringAirFlapBasic; // setpoint from recipe
      L     10; // convert to 0.1%
      *I    ;
      T     "MAL1S032Par".Par.ParIntProcess.PosWitheringAirFlapBasic;
// basic position recycling air to ext. kiln flaps
      L     "MAL1S032Par".StepAct.PosRecycleAirFlapBasic; // setpoint from recipe
      L     10; // convert to 0.1%
      *I    ;
      T     "MAL1S032Par".Par.ParIntProcess.PosBypassExhaustAirFlap;
// basic position recycling air channel flaps
      L     "MAL1S032Par".StepAct.PosWitheringAirFlapBasic; // setpoint from recipe
      L     10; // convert to 0.1%
      *I    ;
      T     "MAL1S032Par".Par.ParIntProcess.PosBypassFreshAirFlap;
// basic position fresh air flaps
//      L     "MAL1S032Par".StepAct.PosFreshAirFlapBasic    // setpoint from recipe
      L     0; // 0%
      U     "MAL1S032Par".Par.FlagProcess.ProcessActive;
      UN    "MAL1S032Par".Par.FlagProcess.Cooling_Activ;
      SPB   klk;
      L     100; // 100%
      U     "MAL1S032Par".Par.FlagProcess.ProcessActive;
      U     "MAL1S032Par".Par.FlagProcess.Cooling_Activ;
      SPB   klk;
      SPA   Nklk;
klk:  L     10; // convert to 0.1%
      *I    ;
      T     "MAL1S032Par".Par.ParIntProcess.PosFreshAirFlapBasic;
Nklk: NOP   0;

// Nachlauf der Brenner
//    U     "GCS7_GrCtrlDB".OutEnable[276]    // G276M Heating Kilningbox
      U     "MAL1S032Par".Par.FlagProcess.ProcessActive;
      UN    "MAL1S032Par".Par.FlagProcess.Cooling_Activ;
      =     "MAL1S032Par".Par.FlagProcess.ProgrammSchwelkenDarren;

      U     "MAL1S032Par".Par.FlagProcess.ProgrammSchwelkenDarren;
      L     S5T#1M;
      SA    T     50; // Nachlauf Brenner

      UN    "MAL1S032Par".Par.FlagProcess.ProgrammSchwelkenDarren;
      U     T     50; // Nachlauf Brenner
      =     "MAL1S032Par".Par.FlagProcess1.HilfsRegler_1_Down;
      =     "MAL1S032Par".Par.FlagProcess1.HilfsRegler_2_Down;
      =     "MAL1S032Par".Par.FlagProcess1.HilfsRegler_3_Down;
      =     "MAL1S032Par".Par.FlagProcess1.HilfsRegler_4_Down;

// Sollwert - Istwert vergleich der Temperatur unter der Horde
      L     "MAL1S032Par".StepAct.TemperaturBelowFloor; // setpoint from SCADA
      L     L#10;
      *D    ;
      T     "MAL1S032Par".Par.ProcessValue.TemperaturBelowFloor;

      U     "SYS_Scan0_Tick1min";
      SPBN  NORM;
//- nur alle x Minuten korrigieren ---
      L     "MAL1S032Par".Par.ProcessValue.CorrInterval;
      +     1;
      T     "MAL1S032Par".Par.ProcessValue.CorrInterval;
      L     2; // Korrekturintervall [min]
      >=I   ;
      SPBN  NORM;
      L     0;
      T     "MAL1S032Par".Par.ProcessValue.CorrInterval;

      L     "MAL1S032Par".Par.ProcessValue.TemperaturBelowFloor;
      L     "G269M".A_3191_BTE01.OutValueUnits; // Real-Value Temperature below floor
      -D    ;
      L     50; // Totband in [0.5°C]
      <=D   ;
      SPB   uebe; // wenn größer keine Korrektur
//- zur Sicherheit nicht mehr als 5.0°C zulassen ---
      L     5.000000e+002; // max. Korrektur !
      L     "MAL1S032Par".Par.ProcessValue_Real.SollwertTempKorr;
      <=R   ;
      SPB   uebe;
      L     "MAL1S032Par".Par.ProcessValue_Real.SollwertTempKorr;
      L     1.000000e+000; // Anpassung an Differenz zwischen den PT100
      +R    ;
      T     "MAL1S032Par".Par.ProcessValue_Real.SollwertTempKorr;
uebe: NOP   0;

      L     "MAL1S032Par".Par.ProcessValue.TemperaturBelowFloor;
      L     "G269M".A_3191_BTE01.OutValueUnits; // Real-Value Temperature below floor
      -D    ;
      L     50; // Totband in [0.5°C]
      >=D   ;
      SPB   unte; // wenn kleier keine Korrektur
//- keine negative Korrektur (führt sonst zu Schwingung) ---
      L     0.000000e+000; // keine negative Korrektur !
      L     "MAL1S032Par".Par.ProcessValue_Real.SollwertTempKorr;
      >=R   ;
      SPB   unte;
      L     1.000000e+000; // Anpassung an Differenz zwischen den PT100
      -R    ;
      T     "MAL1S032Par".Par.ProcessValue_Real.SollwertTempKorr;
unte: NOP   0;

//- bei Schrittbegin noch keine Korrektur ---
NORM: L     "MAL1S032Par".ActTimeStepProcess.SteptimeActMinOverall; // Steptime in min overall
      L     8; // Korrekturverzögerung [min]
      >I    ;
      SPB   SET;
      L     0.000000e+000;
      T     "MAL1S032Par".Par.ProcessValue_Real.SollwertTempKorr;
      L     10; // grossen Wert in Intervallzähler vorladen ...
      T     "MAL1S032Par".Par.ProcessValue.CorrInterval; // ... damit nächster 1MinTick gleich wirksam wird

SET:  NOP   0;
      L     "MAL1S032Par".Par.ProcessValue.TemperaturBelowFloor;
      DTR   ;
      L     "MAL1S032Par".Par.ProcessValue_Real.SollwertTempKorr;
      +R    ;
      T     "MAL1S032Par".Par.ProcessValue_Real.T_SOLL_NORM;
      SPA   M641;
      NOP   0;
//- Korrekturfaktor auf "0" setzen ---
      L     0.000000e+000;
      T     "MAL1S032Par".Par.ProcessValue_Real.SollwertTempKorr;
M641: NOP   0;
      SPA   GCPR;

// GCPRO
// setpoint temperature below floor
      NOP   0; // setpoint fans automatic mode
      L     L#0;
      U     "MAL1S032Par".Par.FlagProcess.Cooling_Activ; // switch over to cooling
      SPB   aut1;
      L     "MAL1S032Par".StepAct.TemperaturBelowFloor; // setpoint from SCADA
aut1: NOP   0;
      DTR   ;
      L     1.000000e+001;
      /R    ;
      T     "MAL1S032Par".Par.ProcessValue_Real.T_SOLL_NORM;
// emergency kiln heating
// fan 1
      U(    ;
      L     2#1;
      L     "MAL1S032Par".RecipeHeader.DeselectVentilator; // emergency regime without fan 1
      ==I   ;
      )     ;
      L     "G269M".A_3191_BTE05.OutValuePc; //AIR TEMPERATURE DIFFUSOR FAN 1 :  temperature in diffusor fan 1
      SPBN  c1R1;
      L     "G269M".A_3191_BTE01.OutValuePc; //AIR TEMPERATURE BELOW FLOOR
      L     "G269M".A_3191_BTE05.OutValuePc; //AIR TEMPERATURE DIFFUSOR FAN 1 :  temperature in diffusor fan 2
      <D    ;
      SPBN  c1R1;
      TAK   ;
c1R1: T     "MAL1S032Par".Par.ParIntProcess.ActValueTemperature_R1;
// fan 2
      U(    ;
      L     2#10;
      L     "MAL1S032Par".RecipeHeader.DeselectVentilator; // emergency regime without fan 2
      ==I   ;
      )     ;
      L     "G269M".A_3191_BTE05.OutValuePc; //AIR TEMPERATURE DIFFUSOR FAN 1 :  temperature in diffusor fan 2
      SPBN  c1R2;
      L     "G269M".A_3191_BTE01.OutValuePc; //AIR TEMPERATURE BELOW FLOOR
      L     "G269M".A_3191_BTE05.OutValuePc; //AIR TEMPERATURE DIFFUSOR FAN 1 :  temperature in diffusor fan 1
      <D    ;
      SPBN  c1R2;
      TAK   ;
c1R2: T     "MAL1S032Par".Par.ParIntProcess.ActValueTemperature_R2;

GCPR: NOP   0;

// cooling down
      L     "MAL1S032Par".StepAct.CoolingDown;
      L     1;
      ==I   ;
      S     "MAL1S032Par".Par.FlagProcess.Cooling_Activ;
E608: NOP   0;

// Abdarr-Betrieb aktiv
      L     "MAL1S032Par".Par.ParIntMachine.ActualStep;
      L     "MAL1S033Par".Par.ParIntMachine.ActualStep;
      >I    ;
      =     "MAL1S032Par".Par.FlagProcess.Abdarr_Betrieb_Aktiv;

NETWORK
TITLE =ASW_6090: calculate heat quantity active kilning

